   1:  PR[91,3] = PR[90,3] + 64.079;
   1:L PR[91] R[100]mm/sec CNT100;
   1:  PR[91,1] = PR[90,1] + 22.475;
   1:  PR[91,2] = PR[90,2] + -8.785;
   1:  PR[91,3] = PR[90,3] + 64.084;
   1:L PR[91] R[100]mm/sec CNT100;
   1:  PR[91,1] = PR[90,1] + 22.742;
   1:  PR[91,2] = PR[90,2] + -8.099;
   1:  PR[91,3] = PR[90,3] + 64.091;
   1:L PR[91] R[100]mm/sec CNT100;
   1:  PR[91,1] = PR[90,1] + 23.009;
   1:  PR[91,2] = PR[90,2] + -7.343;
   1:  PR[91,3] = PR[90,3] + 64.097;
   1:L PR[91] R[100]mm/sec CNT100;
   1:  PR[91,1] = PR[90,1] + 23.209;
   1:  PR[91,2] = PR[90,2] + -6.725;
   1:  PR[91,3] = PR[90,3] + 64.104;
   1:L PR[91] R[100]mm/sec CNT100;
   1:  PR[91,1] = PR[90,1] + 23.430;
   1:  PR[91,2] = PR[90,2] + -5.954;
   1:  PR[91,3] = PR[90,3] + 64.110;
   1:L PR[91] R[100]mm/sec CNT100;
   1:  PR[91,1] = PR[90,1] + 23.593;
   1:  PR[91,2] = PR[90,2] + -5.325;
   1:  PR[91,3] = PR[90,3] + 64.117;
   1:L PR[91] R[100]mm/sec CNT100;
   1:  PR[91,1] = PR[90,1] + 23.768;
   1:  PR[91,2] = PR[90,2] + -4.543;
   1:  PR[91,3] = PR[90,3] + 64.122;
   1:L PR[91] R[100]mm/sec CNT100;
   1:  PR[91,1] = PR[90,1] + 23.893;
   1:  PR[91,2] = PR[90,2] + -3.905;
   1:  PR[91,3] = PR[90,3] + 64.129;
   1:L PR[91] R[100]mm/sec CNT100;
   1:  PR[91,1] = PR[90,1] + 24.021;
   1:  PR[91,2] = PR[90,2] + -3.118;
   1:  PR[91,3] = PR[90,3] + 64.135;
   1:L PR[91] R[100]mm/sec CNT100;
   1:  PR[91,1] = PR[90,1] + 24.176;
   1:  PR[91,2] = PR[90,2] + -1.818;
   1:  PR[91,3] = PR[90,3] + 64.142;
   1:L PR[91] R[100]mm/sec CNT100;
   1:  PR[91,1] = PR[90,1] + 24.237;
   1:  PR[91,2] = PR[90,2] + -1.027;
   1:  PR[91,3] = PR[90,3] + 64.153;
   1:L PR[91] R[100]mm/sec CNT100;
   1:  PR[91,1] = PR[90,1] + 24.280;
   1:  PR[91,2] = PR[90,2] + 0.428;
   1:  PR[91,3] = PR[90,3] + 64.160;
   1:L PR[91] R[100]mm/sec CNT100;
   1:  PR[91,1] = PR[90,1] + 24.237;
   1:  PR[91,2] = PR[90,2] + 1.883;
   1:  PR[91,3] = PR[90,3] + 64.173;
   1:L PR[91] R[100]mm/sec CNT100;
   1:  PR[91,1] = PR[90,1] + 24.189;
   1:  PR[91,2] = PR[90,2] + 2.528;
   1:  PR[91,3] = PR[90,3] + 64.185;
   1:L PR[91] R[100]mm/sec CNT100;
   1:  PR[91,1] = PR[90,1] + 24.108;
   1:  PR[91,2] = PR[90,2] + 3.325;
   1:  PR[91,3] = PR[90,3] + 64.191;
   1:L PR[91] R[100]mm/sec CNT100;
   1:  PR[91,1] = PR[90,1] + 24.021;
   1:  PR[91,2] = PR[90,2] + 3.969;
   1:  PR[91,3] = PR[90,3] + 64.198;
   1:L PR[91] R[100]mm/sec CNT100;
   1:  PR[91,1] = PR[90,1] + 23.893;
   1:  PR[91,2] = PR[90,2] + 4.760;
   1:  PR[91,3] = PR[90,3] + 64.203;
   1:L PR[91] R[100]mm/sec CNT100;
   1:  PR[91,1] = PR[90,1] + 23.768;
   1:  PR[91,2] = PR[90,2] + 5.398;
   1:  PR[91,3] = PR[90,3] + 64.210;
   1:L PR[91] R[100]mm/sec CNT100;
   1:  PR[91,1] = PR[90,1] + 23.593;
   1:  PR[91,2] = PR[90,2] + 6.180;
   1:  PR[91,3] = PR[90,3] + 64.216;
   1:L PR[91] R[100]mm/sec CNT100;
   1:  PR[91,1] = PR[90,1] + 23.430;
   1:  PR[91,2] = PR[90,2] + 6.809;
   1:  PR[91,3] = PR[90,3] + 64.223;
   1:L PR[91] R[100]mm/sec CNT100;
   1:  PR[91,1] = PR[90,1] + 23.209;
   1:  PR[91,2] = PR[90,2] + 7.580;
   1:  PR[91,3] = PR[90,3] + 64.229;
   1:L PR[91] R[100]mm/sec CNT100;
   1:  PR[91,1] = PR[90,1] + 23.009;
   1:  PR[91,2] = PR[90,2] + 8.198;
   1:  PR[91,3] = PR[90,3] + 64.236;
   1:L PR[91] R[100]mm/sec CNT100;
   1:  PR[91,1] = PR[90,1] + 22.742;
   1:  PR[91,2] = PR[90,2] + 8.954;
   1:  PR[91,3] = PR[90,3] + 64.241;
   1:L PR[91] R[100]mm/sec CNT100;
   1:  PR[91,1] = PR[90,1] + 22.475;
   1:  PR[91,2] = PR[90,2] + 9.640;
   1:  PR[91,3] = PR[90,3] + 64.248;
   1:L PR[91] R[100]mm/sec CNT100;
   1:  PR[91,1] = PR[90,1] + 22.195;
   1:  PR[91,2] = PR[90,2] + 10.298;
   1:  PR[91,3] = PR[90,3] + 64.255;
   1:L PR[91] R[100]mm/sec CNT100;
   1:  PR[91,1] = PR[90,1] + 21.924;
   1:  PR[91,2] = PR[90,2] + 10.889;
   1:  PR[91,3] = PR[90,3] + 64.261;
   1:L PR[91] R[100]mm/sec CNT100;
   1:  PR[91,1] = PR[90,1] + 21.569;
   1:  PR[91,2] = PR[90,2] + 11.608;
   1:  PR[91,3] = PR[90,3] + 64.266;
   1:L PR[91] R[100]mm/sec CNT100;
   1:  PR[91,1] = PR[90,1] + 21.263;
   1:  PR[91,2] = PR[90,2] + 12.181;
   1:  PR[91,3] = PR[90,3] + 64.273;
   1:L PR[91] R[100]mm/sec CNT100;
   1:  PR[91,1] = PR[90,1] + 20.865;
   1:  PR[91,2] = PR[90,2] + 12.877;
   1:  PR[91,3] = PR[90,3] + 64.279;
   1:L PR[91] R[100]mm/sec CNT100;
   1:  PR[91,1] = PR[90,1] + 20.526;
   1:  PR[91,2] = PR[90,2] + 13.431;
   1:  PR[91,3] = PR[90,3] + 64.286;
   1:L PR[91] R[100]mm/sec CNT100;
   1:  PR[91,1] = PR[90,1] + 20.088;
   1:  PR[91,2] = PR[90,2] + 14.103;
   1:  PR[91,3] = PR[90,3] + 64.292;
   1:L PR[91] R[100]mm/sec CNT100;
   1:  PR[91,1] = PR[90,1] + 19.667;
   1:  PR[91,2] = PR[90,2] + 14.705;
   1:  PR[91,3] = PR[90,3] + 64.298;
   1:L PR[91] R[100]mm/sec CNT100;
   1:  PR[91,1] = PR[90,1] + 18.834;
   1:  PR[91,2] = PR[90,2] + 15.793;
   1:  PR[91,3] = PR[90,3] + 64.305;
   1:L PR[91] R[100]mm/sec CNT100;
   1:  PR[91,1] = PR[90,1] + 18.322;
   1:  PR[91,2] = PR[90,2] + 16.405;
   1:  PR[91,3] = PR[90,3] + 64.317;
   1:L PR[91] R[100]mm/sec CNT100;
   1:  PR[91,1] = PR[90,1] + 17.890;
   1:  PR[91,2] = PR[90,2] + 16.890;
   1:  PR[91,3] = PR[90,3] + 64.324;
   1:L PR[91] R[100]mm/sec CNT100;
   1:  PR[91,1] = PR[90,1] + 17.342;
   1:  PR[91,2] = PR[90,2] + 17.470;
   1:  PR[91,3] = PR[90,3] + 64.329;
   1:L PR[91] R[100]mm/sec CNT100;
   1:  PR[91,1] = PR[90,1] + 16.339;
   1:  PR[91,2] = PR[90,2] + 18.441;
   1:  PR[91,3] = PR[90,3] + 64.336;
   1:L PR[91] R[100]mm/sec CNT100;
   1:  PR[91,1] = PR[90,1] + 15.830;
   1:  PR[91,2] = PR[90,2] + 18.893;
   1:  PR[91,3] = PR[90,3] + 64.348;
   1:L PR[91] R[100]mm/sec CNT100;
   1:  PR[91,1] = PR[90,1] + 15.235;
   1:  PR[91,2] = PR[90,2] + 19.390;
   1:  PR[91,3] = PR[90,3] + 64.354;
   1:L PR[91] R[100]mm/sec CNT100;
   1:  PR[91,1] = PR[90,1] + 14.747;
   1:  PR[91,2] = PR[90,2] + 19.775;
   1:  PR[91,3] = PR[90,3] + 64.361;
   1:L PR[91] R[100]mm/sec CNT100;
   1:  PR[91,1] = PR[90,1] + 14.129;
   1:  PR[91,2] = PR[90,2] + 20.234;
   1:  PR[91,3] = PR[90,3] + 64.366;
   1:L PR[91] R[100]mm/sec CNT100;
   1:  PR[91,1] = PR[90,1] + 13.076;
   1:  PR[91,2] = PR[90,2] + 20.951;
   1:  PR[91,3] = PR[90,3] + 64.373;
   1:L PR[91] R[100]mm/sec CNT100;
   1:  PR[91,1] = PR[90,1] + 12.442;
   1:  PR[91,2] = PR[90,2] + 21.345;
   1:  PR[91,3] = PR[90,3] + 64.384;
   1:L PR[91] R[100]mm/sec CNT100;
   1:  PR[91,1] = PR[90,1] + 11.218;
   1:  PR[91,2] = PR[90,2] + 22.033;
   1:  PR[91,3] = PR[90,3] + 64.391;
   1:L PR[91] R[100]mm/sec CNT100;
   1:  PR[91,1] = PR[90,1] + 10.609;
   1:  PR[91,2] = PR[90,2] + 22.342;
   1:  PR[91,3] = PR[90,3] + 64.403;
   1:L PR[91] R[100]mm/sec CNT100;
   1:  PR[91,1] = PR[90,1] + 9.972;
   1:  PR[91,2] = PR[90,2] + 22.643;
   1:  PR[91,3] = PR[90,3] + 64.409;
   1:L PR[91] R[100]mm/sec CNT100;
   1:  PR[91,1] = PR[90,1] + 8.677;
   1:  PR[91,2] = PR[90,2] + 23.187;
   1:  PR[91,3] = PR[90,3] + 64.415;
   1:L PR[91] R[100]mm/sec CNT100;
   1:  PR[91,1] = PR[90,1] + 8.017;
   1:  PR[91,2] = PR[90,2] + 23.431;
   1:  PR[91,3] = PR[90,3] + 64.427;
   1:L PR[91] R[100]mm/sec CNT100;
   1:  PR[91,1] = PR[90,1] + 6.765;
   1:  PR[91,2] = PR[90,2] + 23.836;
   1:  PR[91,3] = PR[90,3] + 64.433;
   1:L PR[91] R[100]mm/sec CNT100;
   1:  PR[91,1] = PR[90,1] + 6.027;
   1:  PR[91,2] = PR[90,2] + 24.040;
   1:  PR[91,3] = PR[90,3] + 64.445;
   1:L PR[91] R[100]mm/sec CNT100;
   1:  PR[91,1] = PR[90,1] + 4.710;
   1:  PR[91,2] = PR[90,2] + 24.345;
   1:  PR[91,3] = PR[90,3] + 64.451;
   1:L PR[91] R[100]mm/sec CNT100;
   1:  PR[91,1] = PR[90,1] + 4.050;
   1:  PR[91,2] = PR[90,2] + 24.468;
   1:  PR[91,3] = PR[90,3] + 64.463;
   1:L PR[91] R[100]mm/sec CNT100;
   1:  PR[91,1] = PR[90,1] + 3.290;
   1:  PR[91,2] = PR[90,2] + 24.588;
   1:  PR[91,3] = PR[90,3] + 64.469;
   1:L PR[91] R[100]mm/sec CNT100;
   1:  PR[91,1] = PR[90,1] + 1.949;
   1:  PR[91,2] = PR[90,2] + 24.739;
   1:  PR[91,3] = PR[90,3] + 64.475;
   1:L PR[91] R[100]mm/sec CNT100;
   1:  PR[91,1] = PR[90,1] + 0.649;
   1:  PR[91,2] = PR[90,2] + 24.814;
   1:  PR[91,3] = PR[90,3] + 64.487;
   1:L PR[91] R[100]mm/sec CNT100;
   1:  PR[91,1] = PR[90,1] + -0.121;
   1:  PR[91,2] = PR[90,2] + 24.827;
   1:  PR[91,3] = PR[90,3] + 64.498;
   1:L PR[91] R[100]mm/sec CNT100;
   1:  PR[91,1] = PR[90,1] + -0.841;
   1:  PR[91,2] = PR[90,2] + 24.817;
   1:  PR[91,3] = PR[90,3] + 64.505;
   1:L PR[91] R[100]mm/sec CNT100;
   1:  PR[91,1] = PR[90,1] + -1.512;
   1:  PR[91,2] = PR[90,2] + 24.788;
   1:  PR[91,3] = PR[90,3] + 64.511;
   1:L PR[91] R[100]mm/sec CNT100;
   1:  PR[91,1] = PR[90,1] + -2.912;
   1:  PR[91,2] = PR[90,2] + 24.667;
   1:  PR[91,3] = PR[90,3] + 64.517;
   1:L PR[91] R[100]mm/sec CNT100;
   1:  PR[91,1] = PR[90,1] + -3.618;
   1:  PR[91,2] = PR[90,2] + 24.575;
   1:  PR[91,3] = PR[90,3] + 64.529;
   1:L PR[91] R[100]mm/sec CNT100;
   1:  PR[91,1] = PR[90,1] + -4.905;
   1:  PR[91,2] = PR[90,2] + 24.353;
   1:  PR[91,3] = PR[90,3] + 64.536;
   1:L PR[91] R[100]mm/sec CNT100;
   1:  PR[91,1] = PR[90,1] + -5.654;
   1:  PR[91,2] = PR[90,2] + 24.191;
   1:  PR[91,3] = PR[90,3] + 64.547;
   1:L PR[91] R[100]mm/sec CNT100;
   1:  PR[91,1] = PR[90,1] + -6.967;
   1:  PR[91,2] = PR[90,2] + 23.847;
   1:  PR[91,3] = PR[90,3] + 64.553;
   1:L PR[91] R[100]mm/sec CNT100;
   1:  PR[91,1] = PR[90,1] + -7.599;
   1:  PR[91,2] = PR[90,2] + 23.653;
   1:  PR[91,3] = PR[90,3] + 64.565;
   1:L PR[91] R[100]mm/sec CNT100;
   1:  PR[91,1] = PR[90,1] + -8.919;
   1:  PR[91,2] = PR[90,2] + 23.185;
   1:  PR[91,3] = PR[90,3] + 64.571;
   1:L PR[91] R[100]mm/sec CNT100;
   1:  PR[91,1] = PR[90,1] + -10.180;
   1:  PR[91,2] = PR[90,2] + 22.656;
   1:  PR[91,3] = PR[90,3] + 64.583;
   1:L PR[91] R[100]mm/sec CNT100;
   1:  PR[91,1] = PR[90,1] + -11.461;
   1:  PR[91,2] = PR[90,2] + 22.031;
   1:  PR[91,3] = PR[90,3] + 64.595;
   1:L PR[91] R[100]mm/sec CNT100;
   1:  PR[91,1] = PR[90,1] + -12.678;
   1:  PR[91,2] = PR[90,2] + 21.347;
   1:  PR[91,3] = PR[90,3] + 64.607;
   1:L PR[91] R[100]mm/sec CNT100;
   1:  PR[91,1] = PR[90,1] + -13.854;
   1:  PR[91,2] = PR[90,2] + 20.594;
   1:  PR[91,3] = PR[90,3] + 64.619;
   1:L PR[91] R[100]mm/sec CNT100;
   1:  PR[91,1] = PR[90,1] + -14.988;
   1:  PR[91,2] = PR[90,2] + 19.774;
   1:  PR[91,3] = PR[90,3] + 64.632;
   1:L PR[91] R[100]mm/sec CNT100;
   1:  PR[91,1] = PR[90,1] + -15.529;
   1:  PR[91,2] = PR[90,2] + 19.346;
   1:  PR[91,3] = PR[90,3] + 64.644;
   1:L PR[91] R[100]mm/sec CNT100;
   1:  PR[91,1] = PR[90,1] + -16.536;
   1:  PR[91,2] = PR[90,2] + 18.478;
   1:  PR[91,3] = PR[90,3] + 64.650;
   1:L PR[91] R[100]mm/sec CNT100;
   1:  PR[91,1] = PR[90,1] + -17.118;
   1:  PR[91,2] = PR[90,2] + 17.932;
   1:  PR[91,3] = PR[90,3] + 64.661;
   1:L PR[91] R[100]mm/sec CNT100;
   1:  PR[91,1] = PR[90,1] + -17.577;
   1:  PR[91,2] = PR[90,2] + 17.473;
   1:  PR[91,3] = PR[90,3] + 64.668;
   1:L PR[91] R[100]mm/sec CNT100;
   1:  PR[91,1] = PR[90,1] + -18.125;
   1:  PR[91,2] = PR[90,2] + 16.894;
   1:  PR[91,3] = PR[90,3] + 64.674;
   1:L PR[91] R[100]mm/sec CNT100;
   1:  PR[91,1] = PR[90,1] + -19.010;
   1:  PR[91,2] = PR[90,2] + 15.869;
   1:  PR[91,3] = PR[90,3] + 64.681;
   1:L PR[91] R[100]mm/sec CNT100;
   1:  PR[91,1] = PR[90,1] + -19.478;
   1:  PR[91,2] = PR[90,2] + 15.280;
   1:  PR[91,3] = PR[90,3] + 64.692;
   1:L PR[91] R[100]mm/sec CNT100;
   1:  PR[91,1] = PR[90,1] + -19.955;
   1:  PR[91,2] = PR[90,2] + 14.636;
   1:  PR[91,3] = PR[90,3] + 64.699;
   1:L PR[91] R[100]mm/sec CNT100;
   1:  PR[91,1] = PR[90,1] + -20.326;
   1:  PR[91,2] = PR[90,2] + 14.103;
   1:  PR[91,3] = PR[90,3] + 64.706;
   1:L PR[91] R[100]mm/sec CNT100;
   1:  PR[91,1] = PR[90,1] + -20.764;
   1:  PR[91,2] = PR[90,2] + 13.432;
   1:  PR[91,3] = PR[90,3] + 64.712;
   1:L PR[91] R[100]mm/sec CNT100;
   1:  PR[91,1] = PR[90,1] + -21.104;
   1:  PR[91,2] = PR[90,2] + 12.878;
   1:  PR[91,3] = PR[90,3] + 64.719;
   1:L PR[91] R[100]mm/sec CNT100;
   1:  PR[91,1] = PR[90,1] + -21.488;
   1:  PR[91,2] = PR[90,2] + 12.206;
   1:  PR[91,3] = PR[90,3] + 64.724;
   1:L PR[91] R[100]mm/sec CNT100;
   1:  PR[91,1] = PR[90,1] + -21.794;
   1:  PR[91,2] = PR[90,2] + 11.632;
   1:  PR[91,3] = PR[90,3] + 64.731;
   1:L PR[91] R[100]mm/sec CNT100;
   1:  PR[91,1] = PR[90,1] + -22.160;
   1:  PR[91,2] = PR[90,2] + 10.893;
   1:  PR[91,3] = PR[90,3] + 64.737;
   1:L PR[91] R[100]mm/sec CNT100;
   1:  PR[91,1] = PR[90,1] + -22.689;
   1:  PR[91,2] = PR[90,2] + 9.695;
   1:  PR[91,3] = PR[90,3] + 64.744;
   1:L PR[91] R[100]mm/sec CNT100;
   1:  PR[91,1] = PR[90,1] + -22.981;
   1:  PR[91,2] = PR[90,2] + 8.953;
   1:  PR[91,3] = PR[90,3] + 64.755;
   1:L PR[91] R[100]mm/sec CNT100;
   1:  PR[91,1] = PR[90,1] + -23.248;
   1:  PR[91,2] = PR[90,2] + 8.199;
   1:  PR[91,3] = PR[90,3] + 64.762;
   1:L PR[91] R[100]mm/sec CNT100;
   1:  PR[91,1] = PR[90,1] + -23.447;
   1:  PR[91,2] = PR[90,2] + 7.580;
   1:  PR[91,3] = PR[90,3] + 64.769;
   1:L PR[91] R[100]mm/sec CNT100;
   1:  PR[91,1] = PR[90,1] + -23.669;
   1:  PR[91,2] = PR[90,2] + 6.810;
   1:  PR[91,3] = PR[90,3] + 64.775;
   1:L PR[91] R[100]mm/sec CNT100;
   1:  PR[91,1] = PR[90,1] + -23.831;
   1:  PR[91,2] = PR[90,2] + 6.181;
   1:  PR[91,3] = PR[90,3] + 64.782;
   1:L PR[91] R[100]mm/sec CNT100;
   1:  PR[91,1] = PR[90,1] + -24.006;
   1:  PR[91,2] = PR[90,2] + 5.402;
   1:  PR[91,3] = PR[90,3] + 64.787;
   1:L PR[91] R[100]mm/sec CNT100;
   1:  PR[91,1] = PR[90,1] + -24.238;
   1:  PR[91,2] = PR[90,2] + 4.113;
   1:  PR[91,3] = PR[90,3] + 64.794;
   1:L PR[91] R[100]mm/sec CNT100;
   1:  PR[91,1] = PR[90,1] + -24.347;
   1:  PR[91,2] = PR[90,2] + 3.324;
   1:  PR[91,3] = PR[90,3] + 64.805;
   1:L PR[91] R[100]mm/sec CNT100;
   1:  PR[91,1] = PR[90,1] + -24.428;
   1:  PR[91,2] = PR[90,2] + 2.528;
   1:  PR[91,3] = PR[90,3] + 64.812;
   1:L PR[91] R[100]mm/sec CNT100;
   1:  PR[91,1] = PR[90,1] + -24.476;
   1:  PR[91,2] = PR[90,2] + 1.883;
   1:  PR[91,3] = PR[90,3] + 64.819;
   1:L PR[91] R[100]mm/sec CNT100;
   1:  PR[91,1] = PR[90,1] + -24.519;
   1:  PR[91,2] = PR[90,2] + 0.428;
   1:  PR[91,3] = PR[90,3] + 64.825;
   1:L PR[91] R[100]mm/sec CNT100;
   1:  PR[91,1] = PR[90,1] + -24.476;
   1:  PR[91,2] = PR[90,2] + -1.028;
   1:  PR[91,3] = PR[90,3] + 64.838;
   1:L PR[91] R[100]mm/sec CNT100;
   1:  PR[91,1] = PR[90,1] + -24.428;
   1:  PR[91,2] = PR[90,2] + -1.673;
   1:  PR[91,3] = PR[90,3] + 64.850;
   1:L PR[91] R[100]mm/sec CNT100;
   1:  PR[91,1] = PR[90,1] + -24.346;
   1:  PR[91,2] = PR[90,2] + -2.470;
   1:  PR[91,3] = PR[90,3] + 64.856;
   1:L PR[91] R[100]mm/sec CNT100;
   1:  PR[91,1] = PR[90,1] + -24.260;
   1:  PR[91,2] = PR[90,2] + -3.114;
   1:  PR[91,3] = PR[90,3] + 64.863;
   1:L PR[91] R[100]mm/sec CNT100;
   1:  PR[91,1] = PR[90,1] + -24.131;
   1:  PR[91,2] = PR[90,2] + -3.905;
   1:  PR[91,3] = PR[90,3] + 64.868;
   1:L PR[91] R[100]mm/sec CNT100;
   1:  PR[91,1] = PR[90,1] + -24.007;
   1:  PR[91,2] = PR[90,2] + -4.543;
   1:  PR[91,3] = PR[90,3] + 64.875;
   1:L PR[91] R[100]mm/sec CNT100;
   1:  PR[91,1] = PR[90,1] + -23.832;
   1:  PR[91,2] = PR[90,2] + -5.321;
   1:  PR[91,3] = PR[90,3] + 64.881;
   1:L PR[91] R[100]mm/sec CNT100;
   1:  PR[91,1] = PR[90,1] + -23.484;
   1:  PR[91,2] = PR[90,2] + -6.594;
   1:  PR[91,3] = PR[90,3] + 64.888;
   1:L PR[91] R[100]mm/sec CNT100;
   1:  PR[91,1] = PR[90,1] + -23.446;
   1:  PR[91,2] = PR[90,2] + -6.728;
   1:  PR[91,3] = PR[90,3] + 64.899;
   1:L PR[91] R[100]mm/sec CNT100;
   1:  PR[91,1] = PR[90,1] + -23.248;
   1:  PR[91,2] = PR[90,2] + -7.344;
   1:  PR[91,3] = PR[90,3] + 64.901;
   1:L PR[91] R[100]mm/sec CNT100;
   1:  PR[91,1] = PR[90,1] + -22.981;
   1:  PR[91,2] = PR[90,2] + -8.100;
   1:  PR[91,3] = PR[90,3] + 64.906;
   1:L PR[91] R[100]mm/sec CNT100;
   1:  PR[91,1] = PR[90,1] + -22.745;
   1:  PR[91,2] = PR[90,2] + -8.705;
   1:  PR[91,3] = PR[90,3] + 64.913;
   1:L PR[91] R[100]mm/sec CNT100;
   1:  PR[91,1] = PR[90,1] + -22.433;
   1:  PR[91,2] = PR[90,2] + -9.444;
   1:  PR[91,3] = PR[90,3] + 64.919;
   1:L PR[91] R[100]mm/sec CNT100;
   1:  PR[91,1] = PR[90,1] + -22.162;
   1:  PR[91,2] = PR[90,2] + -10.034;
   1:  PR[91,3] = PR[90,3] + 64.926;
   1:L PR[91] R[100]mm/sec CNT100;
   1:  PR[91,1] = PR[90,1] + -21.807;
   1:  PR[91,2] = PR[90,2] + -10.753;
   1:  PR[91,3] = PR[90,3] + 64.931;
   1:L PR[91] R[100]mm/sec CNT100;
   1:  PR[91,1] = PR[90,1] + -21.501;
   1:  PR[91,2] = PR[90,2] + -11.326;
   1:  PR[91,3] = PR[90,3] + 64.938;
   1:L PR[91] R[100]mm/sec CNT100;
   1:  PR[91,1] = PR[90,1] + -21.104;
   1:  PR[91,2] = PR[90,2] + -12.023;
   1:  PR[91,3] = PR[90,3] + 64.944;
   1:L PR[91] R[100]mm/sec CNT100;
   1:  PR[91,1] = PR[90,1] + -20.764;
   1:  PR[91,2] = PR[90,2] + -12.576;
   1:  PR[91,3] = PR[90,3] + 64.951;
   1:L PR[91] R[100]mm/sec CNT100;
   1:  PR[91,1] = PR[90,1] + -20.326;
   1:  PR[91,2] = PR[90,2] + -13.248;
   1:  PR[91,3] = PR[90,3] + 64.957;
   1:L PR[91] R[100]mm/sec CNT100;
   1:  PR[91,1] = PR[90,1] + -19.955;
   1:  PR[91,2] = PR[90,2] + -13.781;
   1:  PR[91,3] = PR[90,3] + 64.963;
   1:L PR[91] R[100]mm/sec CNT100;
   1:  PR[91,1] = PR[90,1] + -19.478;
   1:  PR[91,2] = PR[90,2] + -14.425;
   1:  PR[91,3] = PR[90,3] + 64.969;
   1:L PR[91] R[100]mm/sec CNT100;
   1:  PR[91,1] = PR[90,1] + -19.010;
   1:  PR[91,2] = PR[90,2] + -15.014;
   1:  PR[91,3] = PR[90,3] + 64.976;
   1:L PR[91] R[100]mm/sec CNT100;
   1:  PR[91,1] = PR[90,1] + -18.125;
   1:  PR[91,2] = PR[90,2] + -16.038;
   1:  PR[91,3] = PR[90,3] + 64.983;
   1:L PR[91] R[100]mm/sec CNT100;
   1:  PR[91,1] = PR[90,1] + -17.577;
   1:  PR[91,2] = PR[90,2] + -16.618;
   1:  PR[91,3] = PR[90,3] + 64.994;
   1:L PR[91] R[100]mm/sec CNT100;
   1:  PR[91,1] = PR[90,1] + -17.118;
   1:  PR[91,2] = PR[90,2] + -17.077;
   1:  PR[91,3] = PR[90,3] + 65.001;
   1:L PR[91] R[100]mm/sec CNT100;
   1:  PR[91,1] = PR[90,1] + -16.536;
   1:  PR[91,2] = PR[90,2] + -17.623;
   1:  PR[91,3] = PR[90,3] + 65.007;
   1:L PR[91] R[100]mm/sec CNT100;
   1:  PR[91,1] = PR[90,1] + -15.529;
   1:  PR[91,2] = PR[90,2] + -18.490;
   1:  PR[91,3] = PR[90,3] + 65.014;
   1:L PR[91] R[100]mm/sec CNT100;
   1:  PR[91,1] = PR[90,1] + -14.988;
   1:  PR[91,2] = PR[90,2] + -18.918;
   1:  PR[91,3] = PR[90,3] + 65.025;
   1:L PR[91] R[100]mm/sec CNT100;
   1:  PR[91,1] = PR[90,1] + -13.854;
   1:  PR[91,2] = PR[90,2] + -19.739;
   1:  PR[91,3] = PR[90,3] + 65.031;
   1:L PR[91] R[100]mm/sec CNT100;
   1:  PR[91,1] = PR[90,1] + -12.684;
   1:  PR[91,2] = PR[90,2] + -20.488;
   1:  PR[91,3] = PR[90,3] + 65.043;
   1:L PR[91] R[100]mm/sec CNT100;
   1:  PR[91,1] = PR[90,1] + -11.461;
   1:  PR[91,2] = PR[90,2] + -21.176;
   1:  PR[91,3] = PR[90,3] + 65.056;
   1:L PR[91] R[100]mm/sec CNT100;
   1:  PR[91,1] = PR[90,1] + -10.207;
   1:  PR[91,2] = PR[90,2] + -21.789;
   1:  PR[91,3] = PR[90,3] + 65.068;
   1:L PR[91] R[100]mm/sec CNT100;
   1:  PR[91,1] = PR[90,1] + -8.919;
   1:  PR[91,2] = PR[90,2] + -22.330;
   1:  PR[91,3] = PR[90,3] + 65.080;
   1:L PR[91] R[100]mm/sec CNT100;
   1:  PR[91,1] = PR[90,1] + -7.599;
   1:  PR[91,2] = PR[90,2] + -22.797;
   1:  PR[91,3] = PR[90,3] + 65.092;
   1:L PR[91] R[100]mm/sec CNT100;
   1:  PR[91,1] = PR[90,1] + -6.967;
   1:  PR[91,2] = PR[90,2] + -22.992;
   1:  PR[91,3] = PR[90,3] + 65.104;
   1:L PR[91] R[100]mm/sec CNT100;
   1:  PR[91,1] = PR[90,1] + -5.654;
   1:  PR[91,2] = PR[90,2] + -23.336;
   1:  PR[91,3] = PR[90,3] + 65.110;
   1:L PR[91] R[100]mm/sec CNT100;
   1:  PR[91,1] = PR[90,1] + -4.905;
   1:  PR[91,2] = PR[90,2] + -23.498;
   1:  PR[91,3] = PR[90,3] + 65.122;
   1:L PR[91] R[100]mm/sec CNT100;
   1:  PR[91,1] = PR[90,1] + -3.618;
   1:  PR[91,2] = PR[90,2] + -23.720;
   1:  PR[91,3] = PR[90,3] + 65.128;
   1:L PR[91] R[100]mm/sec CNT100;
   1:  PR[91,1] = PR[90,1] + -2.908;
   1:  PR[91,2] = PR[90,2] + -23.812;
   1:  PR[91,3] = PR[90,3] + 65.140;
   1:L PR[91] R[100]mm/sec CNT100;
   1:  PR[91,1] = PR[90,1] + -2.288;
   1:  PR[91,2] = PR[90,2] + -23.874;
   1:  PR[91,3] = PR[90,3] + 65.146;
   1:L PR[91] R[100]mm/sec CNT100;
   1:  PR[91,1] = PR[90,1] + -1.515;
   1:  PR[91,2] = PR[90,2] + -23.932;
   1:  PR[91,3] = PR[90,3] + 65.151;
   1:L PR[91] R[100]mm/sec CNT100;
   1:  PR[91,1] = PR[90,1] + -0.841;
   1:  PR[91,2] = PR[90,2] + -23.962;
   1:  PR[91,3] = PR[90,3] + 65.158;
   1:L PR[91] R[100]mm/sec CNT100;
   1:  PR[91,1] = PR[90,1] + -0.124;
   1:  PR[91,2] = PR[90,2] + -23.972;
   1:  PR[91,3] = PR[90,3] + 65.164;
   1:L PR[91] R[100]mm/sec CNT100;
   1:  PR[91] = PR[90];
   1:  PR[91,1] = PR[90,1] + 1.301;
   1:  PR[91,2] = PR[90,2] + -23.931;
   1:  PR[91,3] = PR[90,3] + 66.500;
   1:L PR[91] R[100]mm/sec CNT100;
   1:  PR[91,1] = PR[90,1] + 1.921;
   1:  PR[91,2] = PR[90,2] + -23.887;
   1:  PR[91,3] = PR[90,3] + 65.179;
   1:L PR[91] R[100]mm/sec CNT100;
   1:  PR[91,1] = PR[90,1] + 2.710;
   1:  PR[91,2] = PR[90,2] + -23.807;
   1:  PR[91,3] = PR[90,3] + 65.184;
   1:L PR[91] R[100]mm/sec CNT100;
   1:  PR[91,1] = PR[90,1] + 4.122;
   1:  PR[91,2] = PR[90,2] + -23.601;
   1:  PR[91,3] = PR[90,3] + 65.191;
   1:L PR[91] R[100]mm/sec CNT100;
   1:  PR[91,1] = PR[90,1] + 4.733;
   1:  PR[91,2] = PR[90,2] + -23.485;
   1:  PR[91,3] = PR[90,3] + 65.203;
   1:L PR[91] R[100]mm/sec CNT100;
   1:  PR[91,1] = PR[90,1] + 5.932;
   1:  PR[91,2] = PR[90,2] + -23.209;
   1:  PR[91,3] = PR[90,3] + 65.209;
   1:L PR[91] R[100]mm/sec CNT100;
   1:  PR[91,1] = PR[90,1] + 7.303;
   1:  PR[91,2] = PR[90,2] + -22.816;
   1:  PR[91,3] = PR[90,3] + 65.219;
   1:L PR[91] R[100]mm/sec CNT100;
   1:  PR[91,1] = PR[90,1] + 7.926;
   1:  PR[91,2] = PR[90,2] + -22.607;
   1:  PR[91,3] = PR[90,3] + 65.232;
   1:L PR[91] R[100]mm/sec CNT100;
   1:  PR[91,1] = PR[90,1] + 8.635;
   1:  PR[91,2] = PR[90,2] + -22.348;
   1:  PR[91,3] = PR[90,3] + 65.237;
   1:L PR[91] R[100]mm/sec CNT100;
   1:  PR[91,1] = PR[90,1] + 9.543;
   1:  PR[91,2] = PR[90,2] + -21.976;
   1:  PR[91,3] = PR[90,3] + 65.244;
   1:L PR[91] R[100]mm/sec CNT100;
   1:  PR[91,1] = PR[90,1] + 10.623;
   1:  PR[91,2] = PR[90,2] + -21.480;
   1:  PR[91,3] = PR[90,3] + 65.252;
   1:L PR[91] R[100]mm/sec CNT100;
   1:  PR[91,1] = PR[90,1] + 11.608;
   1:  PR[91,2] = PR[90,2] + -20.967;
   1:  PR[91,3] = PR[90,3] + 65.263;
   1:L PR[91] R[100]mm/sec CNT100;
   1:  PR[91,1] = PR[90,1] + 12.457;
   1:  PR[91,2] = PR[90,2] + -20.481;
   1:  PR[91,3] = PR[90,3] + 65.272;
   1:L PR[91] R[100]mm/sec CNT100;
   1:  PR[91,1] = PR[90,1] + 13.594;
   1:  PR[91,2] = PR[90,2] + -19.754;
   1:  PR[91,3] = PR[90,3] + 65.281;
   1:L PR[91] R[100]mm/sec CNT100;
   1:  PR[91,1] = PR[90,1] + 14.800;
   1:  PR[91,2] = PR[90,2] + -18.879;
   1:  PR[91,3] = PR[90,3] + 65.293;
   1:L PR[91] R[100]mm/sec CNT100;
   1:  PR[91,1] = PR[90,1] + 15.899;
   1:  PR[91,2] = PR[90,2] + -17.977;
   1:  PR[91,3] = PR[90,3] + 65.305;
   1:L PR[91] R[100]mm/sec CNT100;
   1:  PR[91,1] = PR[90,1] + 16.730;
   1:  PR[91,2] = PR[90,2] + -17.219;
   1:  PR[91,3] = PR[90,3] + 65.318;
   1:L PR[91] R[100]mm/sec CNT100;
   1:  PR[91,1] = PR[90,1] + 17.276;
   1:  PR[91,2] = PR[90,2] + -16.682;
   1:  PR[91,3] = PR[90,3] + 65.328;
   1:L PR[91] R[100]mm/sec CNT100;
   1:  PR[91,1] = PR[90,1] + 18.269;
   1:  PR[91,2] = PR[90,2] + -15.609;
   1:  PR[91,3] = PR[90,3] + 65.334;
   1:L PR[91] R[100]mm/sec CNT100;
   1:  PR[91,1] = PR[90,1] + 19.198;
   1:  PR[91,2] = PR[90,2] + -14.478;
   1:  PR[91,3] = PR[90,3] + 65.347;
   1:L PR[91] R[100]mm/sec CNT100;
   1:  PR[91,1] = PR[90,1] + 19.601;
   1:  PR[91,2] = PR[90,2] + -13.940;
   1:  PR[91,3] = PR[90,3] + 65.360;
   1:L PR[91] R[100]mm/sec CNT100;
   1:  PR[91,1] = PR[90,1] + 20.050;
   1:  PR[91,2] = PR[90,2] + -13.304;
   1:  PR[91,3] = PR[90,3] + 65.365;
   1:L PR[91] R[100]mm/sec CNT100;
   1:  PR[91,1] = PR[90,1] + 20.595;
   1:  PR[91,2] = PR[90,2] + -12.465;
   1:  PR[91,3] = PR[90,3] + 65.372;
   1:L PR[91] R[100]mm/sec CNT100;
   1:  PR[91,1] = PR[90,1] + 21.062;
   1:  PR[91,2] = PR[90,2] + -11.675;
   1:  PR[91,3] = PR[90,3] + 65.381;
   1:L PR[91] R[100]mm/sec CNT100;
   1:  PR[91,1] = PR[90,1] + 21.544;
   1:  PR[91,2] = PR[90,2] + -10.800;
   1:  PR[91,3] = PR[90,3] + 65.389;
   1:L PR[91] R[100]mm/sec CNT100;
   1:  PR[91,1] = PR[90,1] + 22.177;
   1:  PR[91,2] = PR[90,2] + -9.483;
   1:  PR[91,3] = PR[90,3] + 65.397;
   1:L PR[91] R[100]mm/sec CNT100;
   1:  PR[91,1] = PR[90,1] + 22.564;
   1:  PR[91,2] = PR[90,2] + -8.559;
   1:  PR[91,3] = PR[90,3] + 65.410;
   1:L PR[91] R[100]mm/sec CNT100;
   1:  PR[91,1] = PR[90,1] + 22.728;
   1:  PR[91,2] = PR[90,2] + -8.138;
   1:  PR[91,3] = PR[90,3] + 65.419;
   1:L PR[91] R[100]mm/sec CNT100;
   1:  PR[91,1] = PR[90,1] + 23.058;
   1:  PR[91,2] = PR[90,2] + -7.193;
   1:  PR[91,3] = PR[90,3] + 65.423;
   1:L PR[91] R[100]mm/sec CNT100;
   1:  PR[91,1] = PR[90,1] + 23.327;
   1:  PR[91,2] = PR[90,2] + -6.316;
   1:  PR[91,3] = PR[90,3] + 65.431;
   1:L PR[91] R[100]mm/sec CNT100;
   1:  PR[91,1] = PR[90,1] + 23.586;
   1:  PR[91,2] = PR[90,2] + -5.352;
   1:  PR[91,3] = PR[90,3] + 65.439;
   1:L PR[91] R[100]mm/sec CNT100;
   1:  PR[91,1] = PR[90,1] + 23.889;
   1:  PR[91,2] = PR[90,2] + -3.923;
   1:  PR[91,3] = PR[90,3] + 65.448;
   1:L PR[91] R[100]mm/sec CNT100;
   1:  PR[91,1] = PR[90,1] + 24.106;
   1:  PR[91,2] = PR[90,2] + -2.481;
   1:  PR[91,3] = PR[90,3] + 65.461;
   1:L PR[91] R[100]mm/sec CNT100;
   1:  PR[91,1] = PR[90,1] + 24.203;
   1:  PR[91,2] = PR[90,2] + -1.490;
   1:  PR[91,3] = PR[90,3] + 65.473;
   1:L PR[91] R[100]mm/sec CNT100;
   1:  PR[91,1] = PR[90,1] + 24.257;
   1:  PR[91,2] = PR[90,2] + -0.574;
   1:  PR[91,3] = PR[90,3] + 65.482;
   1:L PR[91] R[100]mm/sec CNT100;
   1:  PR[91,1] = PR[90,1] + 24.281;
   1:  PR[91,2] = PR[90,2] + 0.430;
   1:  PR[91,3] = PR[90,3] + 65.490;
   1:L PR[91] R[100]mm/sec CNT100;
   1:  PR[91,1] = PR[90,1] + 24.274;
   1:  PR[91,2] = PR[90,2] + 0.882;
   1:  PR[91,3] = PR[90,3] + 65.499;
   1:L PR[91] R[100]mm/sec CNT100;
   1:  PR[91,1] = PR[90,1] + 24.237;
   1:  PR[91,2] = PR[90,2] + 1.885;
   1:  PR[91,3] = PR[90,3] + 65.503;
   1:L PR[91] R[100]mm/sec CNT100;
   1:  PR[91,1] = PR[90,1] + 24.106;
   1:  PR[91,2] = PR[90,2] + 3.339;
   1:  PR[91,3] = PR[90,3] + 65.511;
   1:L PR[91] R[100]mm/sec CNT100;
   1:  PR[91,1] = PR[90,1] + 23.889;
   1:  PR[91,2] = PR[90,2] + 4.783;
   1:  PR[91,3] = PR[90,3] + 65.524;
   1:L PR[91] R[100]mm/sec CNT100;
   1:  PR[91,1] = PR[90,1] + 23.802;
   1:  PR[91,2] = PR[90,2] + 5.225;
   1:  PR[91,3] = PR[90,3] + 65.537;
   1:L PR[91] R[100]mm/sec CNT100;
   1:  PR[91,1] = PR[90,1] + 23.587;
   1:  PR[91,2] = PR[90,2] + 6.203;
   1:  PR[91,3] = PR[90,3] + 65.541;
   1:L PR[91] R[100]mm/sec CNT100;
   1:  PR[91,1] = PR[90,1] + 23.199;
   1:  PR[91,2] = PR[90,2] + 7.611;
   1:  PR[91,3] = PR[90,3] + 65.549;
   1:L PR[91] R[100]mm/sec CNT100;
   1:  PR[91,1] = PR[90,1] + 22.727;
   1:  PR[91,2] = PR[90,2] + 8.994;
   1:  PR[91,3] = PR[90,3] + 65.562;
   1:L PR[91] R[100]mm/sec CNT100;
   1:  PR[91,1] = PR[90,1] + 22.448;
   1:  PR[91,2] = PR[90,2] + 9.703;
   1:  PR[91,3] = PR[90,3] + 65.575;
   1:L PR[91] R[100]mm/sec CNT100;
   1:  PR[91,1] = PR[90,1] + 21.984;
   1:  PR[91,2] = PR[90,2] + 10.758;
   1:  PR[91,3] = PR[90,3] + 65.581;
   1:L PR[91] R[100]mm/sec CNT100;
   1:  PR[91,1] = PR[90,1] + 21.545;
   1:  PR[91,2] = PR[90,2] + 11.652;
   1:  PR[91,3] = PR[90,3] + 65.591;
   1:L PR[91] R[100]mm/sec CNT100;
   1:  PR[91,1] = PR[90,1] + 20.835;
   1:  PR[91,2] = PR[90,2] + 12.928;
   1:  PR[91,3] = PR[90,3] + 65.600;
   1:L PR[91] R[100]mm/sec CNT100;
   1:  PR[91,1] = PR[90,1] + 20.048;
   1:  PR[91,2] = PR[90,2] + 14.161;
   1:  PR[91,3] = PR[90,3] + 65.613;
   1:L PR[91] R[100]mm/sec CNT100;
   1:  PR[91,1] = PR[90,1] + 19.603;
   1:  PR[91,2] = PR[90,2] + 14.793;
   1:  PR[91,3] = PR[90,3] + 65.625;
   1:L PR[91] R[100]mm/sec CNT100;
   1:  PR[91,1] = PR[90,1] + 18.910;
   1:  PR[91,2] = PR[90,2] + 15.698;
   1:  PR[91,3] = PR[90,3] + 65.632;
   1:L PR[91] R[100]mm/sec CNT100;
   1:  PR[91,1] = PR[90,1] + 18.271;
   1:  PR[91,2] = PR[90,2] + 16.462;
   1:  PR[91,3] = PR[90,3] + 65.642;
   1:L PR[91] R[100]mm/sec CNT100;
   1:  PR[91,1] = PR[90,1] + 17.276;
   1:  PR[91,2] = PR[90,2] + 17.537;
   1:  PR[91,3] = PR[90,3] + 65.650;
   1:L PR[91] R[100]mm/sec CNT100;
   1:  PR[91,1] = PR[90,1] + 16.728;
   1:  PR[91,2] = PR[90,2] + 18.076;
   1:  PR[91,3] = PR[90,3] + 65.663;
   1:L PR[91] R[100]mm/sec CNT100;
   1:  PR[91,1] = PR[90,1] + 16.230;
   1:  PR[91,2] = PR[90,2] + 18.539;
   1:  PR[91,3] = PR[90,3] + 65.670;
   1:L PR[91] R[100]mm/sec CNT100;
   1:  PR[91,1] = PR[90,1] + 15.145;
   1:  PR[91,2] = PR[90,2] + 19.462;
   1:  PR[91,3] = PR[90,3] + 65.676;
   1:L PR[91] R[100]mm/sec CNT100;
   1:  PR[91,1] = PR[90,1] + 14.011;
   1:  PR[91,2] = PR[90,2] + 20.318;
   1:  PR[91,3] = PR[90,3] + 65.688;
   1:L PR[91] R[100]mm/sec CNT100;
   1:  PR[91,1] = PR[90,1] + 13.227;
   1:  PR[91,2] = PR[90,2] + 20.851;
   1:  PR[91,3] = PR[90,3] + 65.700;
   1:L PR[91] R[100]mm/sec CNT100;
   1:  PR[91,1] = PR[90,1] + 12.460;
   1:  PR[91,2] = PR[90,2] + 21.334;
   1:  PR[91,3] = PR[90,3] + 65.709;
   1:L PR[91] R[100]mm/sec CNT100;
   1:  PR[91,1] = PR[90,1] + 11.217;
   1:  PR[91,2] = PR[90,2] + 22.034;
   1:  PR[91,3] = PR[90,3] + 65.717;
   1:L PR[91] R[100]mm/sec CNT100;
   1:  PR[91,1] = PR[90,1] + 10.623;
   1:  PR[91,2] = PR[90,2] + 22.336;
   1:  PR[91,3] = PR[90,3] + 65.729;
   1:L PR[91] R[100]mm/sec CNT100;
   1:  PR[91,1] = PR[90,1] + 9.950;
   1:  PR[91,2] = PR[90,2] + 22.653;
   1:  PR[91,3] = PR[90,3] + 65.735;
   1:L PR[91] R[100]mm/sec CNT100;
   1:  PR[91,1] = PR[90,1] + 8.633;
   1:  PR[91,2] = PR[90,2] + 23.204;
   1:  PR[91,3] = PR[90,3] + 65.741;
   1:L PR[91] R[100]mm/sec CNT100;
   1:  PR[91,1] = PR[90,1] + 7.929;
   1:  PR[91,2] = PR[90,2] + 23.461;
   1:  PR[91,3] = PR[90,3] + 65.754;
   1:L PR[91] R[100]mm/sec CNT100;
   1:  PR[91,1] = PR[90,1] + 6.878;
   1:  PR[91,2] = PR[90,2] + 23.802;
   1:  PR[91,3] = PR[90,3] + 65.760;
   1:L PR[91] R[100]mm/sec CNT100;
   1:  PR[91,1] = PR[90,1] + 5.935;
   1:  PR[91,2] = PR[90,2] + 24.064;
   1:  PR[91,3] = PR[90,3] + 65.770;
   1:L PR[91] R[100]mm/sec CNT100;
   1:  PR[91,1] = PR[90,1] + 4.733;
   1:  PR[91,2] = PR[90,2] + 24.340;
   1:  PR[91,3] = PR[90,3] + 65.778;
   1:L PR[91] R[100]mm/sec CNT100;
   1:  PR[91,1] = PR[90,1] + 4.119;
   1:  PR[91,2] = PR[90,2] + 24.456;
   1:  PR[91,3] = PR[90,3] + 65.789;
   1:L PR[91] R[100]mm/sec CNT100;
   1:  PR[91,1] = PR[90,1] + 3.151;
   1:  PR[91,2] = PR[90,2] + 24.606;
   1:  PR[91,3] = PR[90,3] + 65.794;
   1:L PR[91] R[100]mm/sec CNT100;
   1:  PR[91,1] = PR[90,1] + 1.922;
   1:  PR[91,2] = PR[90,2] + 24.742;
   1:  PR[91,3] = PR[90,3] + 65.803;
   1:L PR[91] R[100]mm/sec CNT100;
   1:  PR[91,1] = PR[90,1] + 0.859;
   1:  PR[91,2] = PR[90,2] + 24.805;
   1:  PR[91,3] = PR[90,3] + 65.813;
   1:L PR[91] R[100]mm/sec CNT100;
   1:  PR[91,1] = PR[90,1] + -0.123;
   1:  PR[91,2] = PR[90,2] + 24.827;
   1:  PR[91,3] = PR[90,3] + 65.823;
   1:L PR[91] R[100]mm/sec CNT100;
   1:  PR[91,1] = PR[90,1] + -0.555;
   1:  PR[91,2] = PR[90,2] + 24.821;
   1:  PR[91,3] = PR[90,3] + 65.831;
   1:L PR[91] R[100]mm/sec CNT100;
   1:  PR[91,1] = PR[90,1] + -1.536;
   1:  PR[91,2] = PR[90,2] + 24.786;
   1:  PR[91,3] = PR[90,3] + 65.835;
   1:L PR[91] R[100]mm/sec CNT100;
   1:  PR[91,1] = PR[90,1] + -2.957;
   1:  PR[91,2] = PR[90,2] + 24.662;
   1:  PR[91,3] = PR[90,3] + 65.843;
   1:L PR[91] R[100]mm/sec CNT100;
   1:  PR[91,1] = PR[90,1] + -3.734;
   1:  PR[91,2] = PR[90,2] + 24.557;
   1:  PR[91,3] = PR[90,3] + 65.856;
   1:L PR[91] R[100]mm/sec CNT100;
   1:  PR[91,1] = PR[90,1] + -4.789;
   1:  PR[91,2] = PR[90,2] + 24.375;
   1:  PR[91,3] = PR[90,3] + 65.863;
   1:L PR[91] R[100]mm/sec CNT100;
   1:  PR[91,1] = PR[90,1] + -5.745;
   1:  PR[91,2] = PR[90,2] + 24.169;
   1:  PR[91,3] = PR[90,3] + 65.872;
   1:L PR[91] R[100]mm/sec CNT100;
   1:  PR[91,1] = PR[90,1] + -6.960;
   1:  PR[91,2] = PR[90,2] + 23.849;
   1:  PR[91,3] = PR[90,3] + 65.880;
   1:L PR[91] R[100]mm/sec CNT100;
   1:  PR[91,1] = PR[90,1] + -7.532;
   1:  PR[91,2] = PR[90,2] + 23.674;
   1:  PR[91,3] = PR[90,3] + 65.891;
   1:L PR[91] R[100]mm/sec CNT100;
   1:  PR[91,1] = PR[90,1] + -8.875;
   1:  PR[91,2] = PR[90,2] + 23.202;
   1:  PR[91,3] = PR[90,3] + 65.897;
   1:L PR[91] R[100]mm/sec CNT100;
   1:  PR[91,1] = PR[90,1] + -10.185;
   1:  PR[91,2] = PR[90,2] + 22.654;
   1:  PR[91,3] = PR[90,3] + 65.909;
   1:L PR[91] R[100]mm/sec CNT100;
   1:  PR[91,1] = PR[90,1] + -11.460;
   1:  PR[91,2] = PR[90,2] + 22.032;
   1:  PR[91,3] = PR[90,3] + 65.921;
   1:L PR[91] R[100]mm/sec CNT100;
   1:  PR[91,1] = PR[90,1] + -12.697;
   1:  PR[91,2] = PR[90,2] + 21.336;
   1:  PR[91,3] = PR[90,3] + 65.934;
   1:L PR[91] R[100]mm/sec CNT100;
   1:  PR[91,1] = PR[90,1] + -13.891;
   1:  PR[91,2] = PR[90,2] + 20.569;
   1:  PR[91,3] = PR[90,3] + 65.946;
   1:L PR[91] R[100]mm/sec CNT100;
   1:  PR[91,1] = PR[90,1] + -15.043;
   1:  PR[91,2] = PR[90,2] + 19.731;
   1:  PR[91,3] = PR[90,3] + 65.958;
   1:L PR[91] R[100]mm/sec CNT100;
   1:  PR[91,1] = PR[90,1] + -15.381;
   1:  PR[91,2] = PR[90,2] + 19.464;
   1:  PR[91,3] = PR[90,3] + 65.970;
   1:L PR[91] R[100]mm/sec CNT100;
   1:  PR[91,1] = PR[90,1] + -15.929;
   1:  PR[91,2] = PR[90,2] + 19.011;
   1:  PR[91,3] = PR[90,3] + 65.974;
   1:L PR[91] R[100]mm/sec CNT100;
   1:  PR[91,1] = PR[90,1] + -16.463;
   1:  PR[91,2] = PR[90,2] + 18.544;
   1:  PR[91,3] = PR[90,3] + 65.980;
   1:L PR[91] R[100]mm/sec CNT100;
   1:  PR[91,1] = PR[90,1] + -17.190;
   1:  PR[91,2] = PR[90,2] + 17.860;
   1:  PR[91,3] = PR[90,3] + 65.987;
   1:L PR[91] R[100]mm/sec CNT100;
   1:  PR[91,1] = PR[90,1] + -18.206;
   1:  PR[91,2] = PR[90,2] + 16.803;
   1:  PR[91,3] = PR[90,3] + 65.995;
   1:L PR[91] R[100]mm/sec CNT100;
   1:  PR[91,1] = PR[90,1] + -18.610;
   1:  PR[91,2] = PR[90,2] + 16.347;
   1:  PR[91,3] = PR[90,3] + 66.008;
   1:L PR[91] R[100]mm/sec CNT100;
   1:  PR[91,1] = PR[90,1] + -19.433;
   1:  PR[91,2] = PR[90,2] + 15.338;
   1:  PR[91,3] = PR[90,3] + 66.013;
   1:L PR[91] R[100]mm/sec CNT100;
   1:  PR[91,1] = PR[90,1] + -20.289;
   1:  PR[91,2] = PR[90,2] + 14.158;
   1:  PR[91,3] = PR[90,3] + 66.025;
   1:L PR[91] R[100]mm/sec CNT100;
   1:  PR[91,1] = PR[90,1] + -21.075;
   1:  PR[91,2] = PR[90,2] + 12.925;
   1:  PR[91,3] = PR[90,3] + 66.037;
   1:L PR[91] R[100]mm/sec CNT100;
   1:  PR[91,1] = PR[90,1] + -21.521;
   1:  PR[91,2] = PR[90,2] + 12.145;
   1:  PR[91,3] = PR[90,3] + 66.050;
   1:L PR[91] R[100]mm/sec CNT100;
   1:  PR[91,1] = PR[90,1] + -21.781;
   1:  PR[91,2] = PR[90,2] + 11.657;
   1:  PR[91,3] = PR[90,3] + 66.058;
   1:L PR[91] R[100]mm/sec CNT100;
   1:  PR[91,1] = PR[90,1] + -22.223;
   1:  PR[91,2] = PR[90,2] + 10.758;
   1:  PR[91,3] = PR[90,3] + 66.062;
   1:L PR[91] R[100]mm/sec CNT100;
   1:  PR[91,1] = PR[90,1] + -22.593;
   1:  PR[91,2] = PR[90,2] + 9.919;
   1:  PR[91,3] = PR[90,3] + 66.071;
   1:L PR[91] R[100]mm/sec CNT100;
   1:  PR[91,1] = PR[90,1] + -22.966;
   1:  PR[91,2] = PR[90,2] + 8.992;
   1:  PR[91,3] = PR[90,3] + 66.079;
   1:L PR[91] R[100]mm/sec CNT100;
   1:  PR[91,1] = PR[90,1] + -23.437;
   1:  PR[91,2] = PR[90,2] + 7.611;
   1:  PR[91,3] = PR[90,3] + 66.088;
   1:L PR[91] R[100]mm/sec CNT100;
   1:  PR[91,1] = PR[90,1] + -23.825;
   1:  PR[91,2] = PR[90,2] + 6.203;
   1:  PR[91,3] = PR[90,3] + 66.100;
   1:L PR[91] R[100]mm/sec CNT100;
   1:  PR[91,1] = PR[90,1] + -24.040;
   1:  PR[91,2] = PR[90,2] + 5.229;
   1:  PR[91,3] = PR[90,3] + 66.113;
   1:L PR[91] R[100]mm/sec CNT100;
   1:  PR[91,1] = PR[90,1] + -24.202;
   1:  PR[91,2] = PR[90,2] + 4.326;
   1:  PR[91,3] = PR[90,3] + 66.122;
   1:L PR[91] R[100]mm/sec CNT100;
   1:  PR[91,1] = PR[90,1] + -24.344;
   1:  PR[91,2] = PR[90,2] + 3.341;
   1:  PR[91,3] = PR[90,3] + 66.130;
   1:L PR[91] R[100]mm/sec CNT100;
   1:  PR[91,1] = PR[90,1] + -24.475;
   1:  PR[91,2] = PR[90,2] + 1.887;
   1:  PR[91,3] = PR[90,3] + 66.138;
   1:L PR[91] R[100]mm/sec CNT100;
   1:  PR[91,1] = PR[90,1] + -24.519;
   1:  PR[91,2] = PR[90,2] + 0.428;
   1:  PR[91,3] = PR[90,3] + 66.151;
   1:L PR[91] R[100]mm/sec CNT100;
   1:  PR[91,1] = PR[90,1] + -24.475;
   1:  PR[91,2] = PR[90,2] + -1.037;
   1:  PR[91,3] = PR[90,3] + 66.164;
   1:L PR[91] R[100]mm/sec CNT100;
   1:  PR[91,1] = PR[90,1] + -24.442;
   1:  PR[91,2] = PR[90,2] + -1.485;
   1:  PR[91,3] = PR[90,3] + 66.176;
   1:L PR[91] R[100]mm/sec CNT100;
   1:  PR[91,1] = PR[90,1] + -24.345;
   1:  PR[91,2] = PR[90,2] + -2.482;
   1:  PR[91,3] = PR[90,3] + 66.180;
   1:L PR[91] R[100]mm/sec CNT100;
   1:  PR[91,1] = PR[90,1] + -24.128;
   1:  PR[91,2] = PR[90,2] + -3.923;
   1:  PR[91,3] = PR[90,3] + 66.189;
   1:L PR[91] R[100]mm/sec CNT100;
   1:  PR[91,1] = PR[90,1] + -23.825;
   1:  PR[91,2] = PR[90,2] + -5.351;
   1:  PR[91,3] = PR[90,3] + 66.202;
   1:L PR[91] R[100]mm/sec CNT100;
   1:  PR[91,1] = PR[90,1] + -23.581;
   1:  PR[91,2] = PR[90,2] + -6.240;
   1:  PR[91,3] = PR[90,3] + 66.214;
   1:L PR[91] R[100]mm/sec CNT100;
   1:  PR[91,1] = PR[90,1] + -23.438;
   1:  PR[91,2] = PR[90,2] + -6.755;
   1:  PR[91,3] = PR[90,3] + 66.222;
   1:L PR[91] R[100]mm/sec CNT100;
   1:  PR[91,1] = PR[90,1] + -22.967;
   1:  PR[91,2] = PR[90,2] + -8.135;
   1:  PR[91,3] = PR[90,3] + 66.227;
   1:L PR[91] R[100]mm/sec CNT100;
   1:  PR[91,1] = PR[90,1] + -22.414;
   1:  PR[91,2] = PR[90,2] + -9.486;
   1:  PR[91,3] = PR[90,3] + 66.240;
   1:L PR[91] R[100]mm/sec CNT100;
   1:  PR[91,1] = PR[90,1] + -21.780;
   1:  PR[91,2] = PR[90,2] + -10.804;
   1:  PR[91,3] = PR[90,3] + 66.252;
   1:L PR[91] R[100]mm/sec CNT100;
   1:  PR[91,1] = PR[90,1] + -21.521;
   1:  PR[91,2] = PR[90,2] + -11.289;
   1:  PR[91,3] = PR[90,3] + 66.265;
   1:L PR[91] R[100]mm/sec CNT100;
   1:  PR[91,1] = PR[90,1] + -21.075;
   1:  PR[91,2] = PR[90,2] + -12.070;
   1:  PR[91,3] = PR[90,3] + 66.270;
   1:L PR[91] R[100]mm/sec CNT100;
   1:  PR[91,1] = PR[90,1] + -20.289;
   1:  PR[91,2] = PR[90,2] + -13.303;
   1:  PR[91,3] = PR[90,3] + 66.278;
   1:L PR[91] R[100]mm/sec CNT100;
   1:  PR[91,1] = PR[90,1] + -19.431;
   1:  PR[91,2] = PR[90,2] + -14.485;
   1:  PR[91,3] = PR[90,3] + 66.290;
   1:L PR[91] R[100]mm/sec CNT100;
   1:  PR[91,1] = PR[90,1] + -18.908;
   1:  PR[91,2] = PR[90,2] + -15.137;
   1:  PR[91,3] = PR[90,3] + 66.303;
   1:L PR[91] R[100]mm/sec CNT100;
   1:  PR[91,1] = PR[90,1] + -18.204;
   1:  PR[91,2] = PR[90,2] + -15.950;
   1:  PR[91,3] = PR[90,3] + 66.310;
   1:L PR[91] R[100]mm/sec CNT100;
   1:  PR[91,1] = PR[90,1] + -17.190;
   1:  PR[91,2] = PR[90,2] + -17.005;
   1:  PR[91,3] = PR[90,3] + 66.319;
   1:L PR[91] R[100]mm/sec CNT100;
   1:  PR[91,1] = PR[90,1] + -16.465;
   1:  PR[91,2] = PR[90,2] + -17.687;
   1:  PR[91,3] = PR[90,3] + 66.332;
   1:L PR[91] R[100]mm/sec CNT100;
   1:  PR[91,1] = PR[90,1] + -15.590;
   1:  PR[91,2] = PR[90,2] + -18.440;
   1:  PR[91,3] = PR[90,3] + 66.341;
   1:L PR[91] R[100]mm/sec CNT100;
   1:  PR[91,1] = PR[90,1] + -15.042;
   1:  PR[91,2] = PR[90,2] + -18.877;
   1:  PR[91,3] = PR[90,3] + 66.351;
   1:L PR[91] R[100]mm/sec CNT100;
   1:  PR[91,1] = PR[90,1] + -13.891;
   1:  PR[91,2] = PR[90,2] + -19.714;
   1:  PR[91,3] = PR[90,3] + 66.357;
   1:L PR[91] R[100]mm/sec CNT100;
   1:  PR[91,1] = PR[90,1] + -12.718;
   1:  PR[91,2] = PR[90,2] + -20.468;
   1:  PR[91,3] = PR[90,3] + 66.369;
   1:L PR[91] R[100]mm/sec CNT100;
   1:  PR[91,1] = PR[90,1] + -11.460;
   1:  PR[91,2] = PR[90,2] + -21.177;
   1:  PR[91,3] = PR[90,3] + 66.381;
   1:L PR[91] R[100]mm/sec CNT100;
   1:  PR[91,1] = PR[90,1] + -10.185;
   1:  PR[91,2] = PR[90,2] + -21.799;
   1:  PR[91,3] = PR[90,3] + 66.394;
   1:L PR[91] R[100]mm/sec CNT100;
   1:  PR[91,1] = PR[90,1] + -8.875;
   1:  PR[91,2] = PR[90,2] + -22.347;
   1:  PR[91,3] = PR[90,3] + 66.406;
   1:L PR[91] R[100]mm/sec CNT100;
   1:  PR[91,1] = PR[90,1] + -7.532;
   1:  PR[91,2] = PR[90,2] + -22.819;
   1:  PR[91,3] = PR[90,3] + 66.418;
   1:L PR[91] R[100]mm/sec CNT100;
   1:  PR[91,1] = PR[90,1] + -6.960;
   1:  PR[91,2] = PR[90,2] + -22.994;
   1:  PR[91,3] = PR[90,3] + 66.431;
   1:L PR[91] R[100]mm/sec CNT100;
   1:  PR[91,1] = PR[90,1] + -5.748;
   1:  PR[91,2] = PR[90,2] + -23.313;
   1:  PR[91,3] = PR[90,3] + 66.436;
   1:L PR[91] R[100]mm/sec CNT100;
   1:  PR[91,1] = PR[90,1] + -4.356;
   1:  PR[91,2] = PR[90,2] + -23.601;
   1:  PR[91,3] = PR[90,3] + 66.447;
   1:L PR[91] R[100]mm/sec CNT100;
   1:  PR[91,1] = PR[90,1] + -2.951;
   1:  PR[91,2] = PR[90,2] + -23.807;
   1:  PR[91,3] = PR[90,3] + 66.459;
   1:L PR[91] R[100]mm/sec CNT100;
   1:  PR[91,1] = PR[90,1] + -1.977;
   1:  PR[91,2] = PR[90,2] + -23.900;
   1:  PR[91,3] = PR[90,3] + 66.472;
   1:L PR[91] R[100]mm/sec CNT100;
   1:  PR[91,1] = PR[90,1] + -0.911;
   1:  PR[91,2] = PR[90,2] + -23.959;
   1:  PR[91,3] = PR[90,3] + 66.480;
   1:L PR[91] R[100]mm/sec CNT100;
   1:  PR[91,1] = PR[90,1] + 0.321;
   1:  PR[91,2] = PR[90,2] + -23.966;
   1:  PR[91,3] = PR[90,3] + 66.489;
   1:L PR[91] R[100]mm/sec CNT100;
   1:  PR[91] = PR[90];
   1:  PR[91,1] = PR[90,1] + 1.327;
   1:  PR[91,2] = PR[90,2] + -23.929;
   1:  PR[91,3] = PR[90,3] + 67.830;
   1:L PR[91] R[100]mm/sec CNT100;
   1:  PR[91,1] = PR[90,1] + 1.891;
   1:  PR[91,2] = PR[90,2] + -23.889;
   1:  PR[91,3] = PR[90,3] + 66.513;
   1:L PR[91] R[100]mm/sec CNT100;
   1:  PR[91,1] = PR[90,1] + 3.010;
   1:  PR[91,2] = PR[90,2] + -23.769;
   1:  PR[91,3] = PR[90,3] + 66.517;
   1:L PR[91] R[100]mm/sec CNT100;
   1:  PR[91,1] = PR[90,1] + 4.436;
   1:  PR[91,2] = PR[90,2] + -23.542;
   1:  PR[91,3] = PR[90,3] + 66.527;
   1:L PR[91] R[100]mm/sec CNT100;
   1:  PR[91,1] = PR[90,1] + 5.595;
   1:  PR[91,2] = PR[90,2] + -23.293;
   1:  PR[91,3] = PR[90,3] + 66.540;
   1:L PR[91] R[100]mm/sec CNT100;
   1:  PR[91,1] = PR[90,1] + 6.992;
   1:  PR[91,2] = PR[90,2] + -22.912;
   1:  PR[91,3] = PR[90,3] + 66.550;
   1:L PR[91] R[100]mm/sec CNT100;
   1:  PR[91,1] = PR[90,1] + 7.839;
   1:  PR[91,2] = PR[90,2] + -22.637;
   1:  PR[91,3] = PR[90,3] + 66.563;
   1:L PR[91] R[100]mm/sec CNT100;
   1:  PR[91,1] = PR[90,1] + 8.828;
   1:  PR[91,2] = PR[90,2] + -22.269;
   1:  PR[91,3] = PR[90,3] + 66.570;
   1:L PR[91] R[100]mm/sec CNT100;
   1:  PR[91,1] = PR[90,1] + 9.928;
   1:  PR[91,2] = PR[90,2] + -21.807;
   1:  PR[91,3] = PR[90,3] + 66.580;
   1:L PR[91] R[100]mm/sec CNT100;
   1:  PR[91,1] = PR[90,1] + 10.637;
   1:  PR[91,2] = PR[90,2] + -21.474;
   1:  PR[91,3] = PR[90,3] + 66.590;
   1:L PR[91] R[100]mm/sec CNT100;
   1:  PR[91,1] = PR[90,1] + 11.216;
   1:  PR[91,2] = PR[90,2] + -21.180;
   1:  PR[91,3] = PR[90,3] + 66.597;
   1:L PR[91] R[100]mm/sec CNT100;
   1:  PR[91,1] = PR[90,1] + 12.479;
   1:  PR[91,2] = PR[90,2] + -20.468;
   1:  PR[91,3] = PR[90,3] + 66.602;
   1:L PR[91] R[100]mm/sec CNT100;
   1:  PR[91,1] = PR[90,1] + 13.379;
   1:  PR[91,2] = PR[90,2] + -19.896;
   1:  PR[91,3] = PR[90,3] + 66.615;
   1:L PR[91] R[100]mm/sec CNT100;
   1:  PR[91,1] = PR[90,1] + 13.896;
   1:  PR[91,2] = PR[90,2] + -19.544;
   1:  PR[91,3] = PR[90,3] + 66.624;
   1:L PR[91] R[100]mm/sec CNT100;
   1:  PR[91,1] = PR[90,1] + 15.053;
   1:  PR[91,2] = PR[90,2] + -18.680;
   1:  PR[91,3] = PR[90,3] + 66.630;
   1:L PR[91] R[100]mm/sec CNT100;
   1:  PR[91,1] = PR[90,1] + 16.161;
   1:  PR[91,2] = PR[90,2] + -17.746;
   1:  PR[91,3] = PR[90,3] + 66.642;
   1:L PR[91] R[100]mm/sec CNT100;
   1:  PR[91,1] = PR[90,1] + 16.640;
   1:  PR[91,2] = PR[90,2] + -17.305;
   1:  PR[91,3] = PR[90,3] + 66.655;
   1:L PR[91] R[100]mm/sec CNT100;
   1:  PR[91,1] = PR[90,1] + 17.215;
   1:  PR[91,2] = PR[90,2] + -16.743;
   1:  PR[91,3] = PR[90,3] + 66.660;
   1:L PR[91] R[100]mm/sec CNT100;
   1:  PR[91,1] = PR[90,1] + 18.217;
   1:  PR[91,2] = PR[90,2] + -15.669;
   1:  PR[91,3] = PR[90,3] + 66.667;
   1:L PR[91] R[100]mm/sec CNT100;
   1:  PR[91,1] = PR[90,1] + 18.987;
   1:  PR[91,2] = PR[90,2] + -14.747;
   1:  PR[91,3] = PR[90,3] + 66.680;
   1:L PR[91] R[100]mm/sec CNT100;
   1:  PR[91,1] = PR[90,1] + 19.539;
   1:  PR[91,2] = PR[90,2] + -14.025;
   1:  PR[91,3] = PR[90,3] + 66.690;
   1:L PR[91] R[100]mm/sec CNT100;
   1:  PR[91,1] = PR[90,1] + 20.011;
   1:  PR[91,2] = PR[90,2] + -13.361;
   1:  PR[91,3] = PR[90,3] + 66.698;
   1:L PR[91] R[100]mm/sec CNT100;
   1:  PR[91,1] = PR[90,1] + 20.805;
   1:  PR[91,2] = PR[90,2] + -12.123;
   1:  PR[91,3] = PR[90,3] + 66.705;
   1:L PR[91] R[100]mm/sec CNT100;
   1:  PR[91,1] = PR[90,1] + 21.394;
   1:  PR[91,2] = PR[90,2] + -11.082;
   1:  PR[91,3] = PR[90,3] + 66.718;
   1:L PR[91] R[100]mm/sec CNT100;
   1:  PR[91,1] = PR[90,1] + 22.047;
   1:  PR[91,2] = PR[90,2] + -9.767;
   1:  PR[91,3] = PR[90,3] + 66.729;
   1:L PR[91] R[100]mm/sec CNT100;
   1:  PR[91,1] = PR[90,1] + 22.421;
   1:  PR[91,2] = PR[90,2] + -8.915;
   1:  PR[91,3] = PR[90,3] + 66.741;
   1:L PR[91] R[100]mm/sec CNT100;
   1:  PR[91,1] = PR[90,1] + 22.713;
   1:  PR[91,2] = PR[90,2] + -8.176;
   1:  PR[91,3] = PR[90,3] + 66.749;
   1:L PR[91] R[100]mm/sec CNT100;
   1:  PR[91,1] = PR[90,1] + 23.189;
   1:  PR[91,2] = PR[90,2] + -6.788;
   1:  PR[91,3] = PR[90,3] + 66.756;
   1:L PR[91] R[100]mm/sec CNT100;
   1:  PR[91,1] = PR[90,1] + 23.580;
   1:  PR[91,2] = PR[90,2] + -5.375;
   1:  PR[91,3] = PR[90,3] + 66.769;
   1:L PR[91] R[100]mm/sec CNT100;
   1:  PR[91,1] = PR[90,1] + 23.836;
   1:  PR[91,2] = PR[90,2] + -4.201;
   1:  PR[91,3] = PR[90,3] + 66.782;
   1:L PR[91] R[100]mm/sec CNT100;
   1:  PR[91,1] = PR[90,1] + 23.929;
   1:  PR[91,2] = PR[90,2] + -3.684;
   1:  PR[91,3] = PR[90,3] + 66.792;
   1:L PR[91] R[100]mm/sec CNT100;
   1:  PR[91,1] = PR[90,1] + 24.105;
   1:  PR[91,2] = PR[90,2] + -2.497;
   1:  PR[91,3] = PR[90,3] + 66.797;
   1:L PR[91] R[100]mm/sec CNT100;
   1:  PR[91,1] = PR[90,1] + 24.217;
   1:  PR[91,2] = PR[90,2] + -1.302;
   1:  PR[91,3] = PR[90,3] + 66.807;
   1:L PR[91] R[100]mm/sec CNT100;
   1:  PR[91,1] = PR[90,1] + 24.248;
   1:  PR[91,2] = PR[90,2] + -0.778;
   1:  PR[91,3] = PR[90,3] + 66.818;
   1:L PR[91] R[100]mm/sec CNT100;
   1:  PR[91,1] = PR[90,1] + 24.281;
   1:  PR[91,2] = PR[90,2] + 0.427;
   1:  PR[91,3] = PR[90,3] + 66.822;
   1:L PR[91] R[100]mm/sec CNT100;
   1:  PR[91,1] = PR[90,1] + 24.236;
   1:  PR[91,2] = PR[90,2] + 1.895;
   1:  PR[91,3] = PR[90,3] + 66.833;
   1:L PR[91] R[100]mm/sec CNT100;
   1:  PR[91,1] = PR[90,1] + 24.104;
   1:  PR[91,2] = PR[90,2] + 3.353;
   1:  PR[91,3] = PR[90,3] + 66.845;
   1:L PR[91] R[100]mm/sec CNT100;
   1:  PR[91,1] = PR[90,1] + 23.886;
   1:  PR[91,2] = PR[90,2] + 4.796;
   1:  PR[91,3] = PR[90,3] + 66.858;
   1:L PR[91] R[100]mm/sec CNT100;
   1:  PR[91,1] = PR[90,1] + 23.513;
   1:  PR[91,2] = PR[90,2] + 6.492;
   1:  PR[91,3] = PR[90,3] + 66.871;
   1:L PR[91] R[100]mm/sec CNT100;
   1:  PR[91,1] = PR[90,1] + 23.189;
   1:  PR[91,2] = PR[90,2] + 7.642;
   1:  PR[91,3] = PR[90,3] + 66.886;
   1:L PR[91] R[100]mm/sec CNT100;
   1:  PR[91,1] = PR[90,1] + 22.713;
   1:  PR[91,2] = PR[90,2] + 9.031;
   1:  PR[91,3] = PR[90,3] + 66.896;
   1:L PR[91] R[100]mm/sec CNT100;
   1:  PR[91,1] = PR[90,1] + 22.421;
   1:  PR[91,2] = PR[90,2] + 9.770;
   1:  PR[91,3] = PR[90,3] + 66.909;
   1:L PR[91] R[100]mm/sec CNT100;
   1:  PR[91,1] = PR[90,1] + 22.046;
   1:  PR[91,2] = PR[90,2] + 10.624;
   1:  PR[91,3] = PR[90,3] + 66.916;
   1:L PR[91] R[100]mm/sec CNT100;
   1:  PR[91,1] = PR[90,1] + 21.520;
   1:  PR[91,2] = PR[90,2] + 11.700;
   1:  PR[91,3] = PR[90,3] + 66.924;
   1:L PR[91] R[100]mm/sec CNT100;
   1:  PR[91,1] = PR[90,1] + 20.804;
   1:  PR[91,2] = PR[90,2] + 12.979;
   1:  PR[91,3] = PR[90,3] + 66.934;
   1:L PR[91] R[100]mm/sec CNT100;
   1:  PR[91,1] = PR[90,1] + 20.011;
   1:  PR[91,2] = PR[90,2] + 14.215;
   1:  PR[91,3] = PR[90,3] + 66.947;
   1:L PR[91] R[100]mm/sec CNT100;
   1:  PR[91,1] = PR[90,1] + 19.378;
   1:  PR[91,2] = PR[90,2] + 15.097;
   1:  PR[91,3] = PR[90,3] + 66.960;
   1:L PR[91] R[100]mm/sec CNT100;
   1:  PR[91,1] = PR[90,1] + 18.989;
   1:  PR[91,2] = PR[90,2] + 15.599;
   1:  PR[91,3] = PR[90,3] + 66.969;
   1:L PR[91] R[100]mm/sec CNT100;
   1:  PR[91,1] = PR[90,1] + 18.038;
   1:  PR[91,2] = PR[90,2] + 16.725;
   1:  PR[91,3] = PR[90,3] + 66.975;
   1:L PR[91] R[100]mm/sec CNT100;
   1:  PR[91,1] = PR[90,1] + 17.216;
   1:  PR[91,2] = PR[90,2] + 17.597;
   1:  PR[91,3] = PR[90,3] + 66.987;
   1:L PR[91] R[100]mm/sec CNT100;
   1:  PR[91,1] = PR[90,1] + 16.640;
   1:  PR[91,2] = PR[90,2] + 18.160;
   1:  PR[91,3] = PR[90,3] + 66.998;
   1:L PR[91] R[100]mm/sec CNT100;
   1:  PR[91,1] = PR[90,1] + 16.160;
   1:  PR[91,2] = PR[90,2] + 18.601;
   1:  PR[91,3] = PR[90,3] + 67.005;
   1:L PR[91] R[100]mm/sec CNT100;
   1:  PR[91,1] = PR[90,1] + 15.050;
   1:  PR[91,2] = PR[90,2] + 19.537;
   1:  PR[91,3] = PR[90,3] + 67.010;
   1:L PR[91] R[100]mm/sec CNT100;
   1:  PR[91,1] = PR[90,1] + 14.654;
   1:  PR[91,2] = PR[90,2] + 19.841;
   1:  PR[91,3] = PR[90,3] + 67.023;
   1:L PR[91] R[100]mm/sec CNT100;
   1:  PR[91,1] = PR[90,1] + 13.589;
   1:  PR[91,2] = PR[90,2] + 20.613;
   1:  PR[91,3] = PR[90,3] + 67.027;
   1:L PR[91] R[100]mm/sec CNT100;
   1:  PR[91,1] = PR[90,1] + 12.478;
   1:  PR[91,2] = PR[90,2] + 21.324;
   1:  PR[91,3] = PR[90,3] + 67.039;
   1:L PR[91] R[100]mm/sec CNT100;
   1:  PR[91,1] = PR[90,1] + 11.216;
   1:  PR[91,2] = PR[90,2] + 22.035;
   1:  PR[91,3] = PR[90,3] + 67.050;
   1:L PR[91] R[100]mm/sec CNT100;
   1:  PR[91,1] = PR[90,1] + 10.637;
   1:  PR[91,2] = PR[90,2] + 22.329;
   1:  PR[91,3] = PR[90,3] + 67.063;
   1:L PR[91] R[100]mm/sec CNT100;
   1:  PR[91,1] = PR[90,1] + 9.929;
   1:  PR[91,2] = PR[90,2] + 22.662;
   1:  PR[91,3] = PR[90,3] + 67.068;
   1:L PR[91] R[100]mm/sec CNT100;
   1:  PR[91,1] = PR[90,1] + 8.589;
   1:  PR[91,2] = PR[90,2] + 23.220;
   1:  PR[91,3] = PR[90,3] + 67.075;
   1:L PR[91] R[100]mm/sec CNT100;
   1:  PR[91,1] = PR[90,1] + 7.841;
   1:  PR[91,2] = PR[90,2] + 23.492;
   1:  PR[91,3] = PR[90,3] + 67.088;
   1:L PR[91] R[100]mm/sec CNT100;
   1:  PR[91,1] = PR[90,1] + 6.992;
   1:  PR[91,2] = PR[90,2] + 23.767;
   1:  PR[91,3] = PR[90,3] + 67.095;
   1:L PR[91] R[100]mm/sec CNT100;
   1:  PR[91,1] = PR[90,1] + 5.593;
   1:  PR[91,2] = PR[90,2] + 24.148;
   1:  PR[91,3] = PR[90,3] + 67.102;
   1:L PR[91] R[100]mm/sec CNT100;
   1:  PR[91,1] = PR[90,1] + 4.756;
   1:  PR[91,2] = PR[90,2] + 24.335;
   1:  PR[91,3] = PR[90,3] + 67.115;
   1:L PR[91] R[100]mm/sec CNT100;
   1:  PR[91,1] = PR[90,1] + 4.189;
   1:  PR[91,2] = PR[90,2] + 24.444;
   1:  PR[91,3] = PR[90,3] + 67.122;
   1:L PR[91] R[100]mm/sec CNT100;
   1:  PR[91,1] = PR[90,1] + 3.012;
   1:  PR[91,2] = PR[90,2] + 24.624;
   1:  PR[91,3] = PR[90,3] + 67.127;
   1:L PR[91] R[100]mm/sec CNT100;
   1:  PR[91,1] = PR[90,1] + 1.894;
   1:  PR[91,2] = PR[90,2] + 24.744;
   1:  PR[91,3] = PR[90,3] + 67.138;
   1:L PR[91] R[100]mm/sec CNT100;
   1:  PR[91,1] = PR[90,1] + 1.069;
   1:  PR[91,2] = PR[90,2] + 24.795;
   1:  PR[91,3] = PR[90,3] + 67.148;
   1:L PR[91] R[100]mm/sec CNT100;
   1:  PR[91,1] = PR[90,1] + -0.122;
   1:  PR[91,2] = PR[90,2] + 24.827;
   1:  PR[91,3] = PR[90,3] + 67.155;
   1:L PR[91] R[100]mm/sec CNT100;
   1:  PR[91,1] = PR[90,1] + -0.980;
   1:  PR[91,2] = PR[90,2] + 24.812;
   1:  PR[91,3] = PR[90,3] + 67.165;
   1:L PR[91] R[100]mm/sec CNT100;
   1:  PR[91,1] = PR[90,1] + -1.556;
   1:  PR[91,2] = PR[90,2] + 24.785;
   1:  PR[91,3] = PR[90,3] + 67.173;
   1:L PR[91] R[100]mm/sec CNT100;
   1:  PR[91,1] = PR[90,1] + -3.002;
   1:  PR[91,2] = PR[90,2] + 24.656;
   1:  PR[91,3] = PR[90,3] + 67.178;
   1:L PR[91] R[100]mm/sec CNT100;
   1:  PR[91,1] = PR[90,1] + -3.850;
   1:  PR[91,2] = PR[90,2] + 24.540;
   1:  PR[91,3] = PR[90,3] + 67.190;
   1:L PR[91] R[100]mm/sec CNT100;
   1:  PR[91,1] = PR[90,1] + -4.670;
   1:  PR[91,2] = PR[90,2] + 24.398;
   1:  PR[91,3] = PR[90,3] + 67.198;
   1:L PR[91] R[100]mm/sec CNT100;
   1:  PR[91,1] = PR[90,1] + -6.086;
   1:  PR[91,2] = PR[90,2] + 24.086;
   1:  PR[91,3] = PR[90,3] + 67.205;
   1:L PR[91] R[100]mm/sec CNT100;
   1:  PR[91,1] = PR[90,1] + -6.952;
   1:  PR[91,2] = PR[90,2] + 23.851;
   1:  PR[91,3] = PR[90,3] + 67.217;
   1:L PR[91] R[100]mm/sec CNT100;
   1:  PR[91,1] = PR[90,1] + -7.465;
   1:  PR[91,2] = PR[90,2] + 23.695;
   1:  PR[91,3] = PR[90,3] + 67.225;
   1:L PR[91] R[100]mm/sec CNT100;
   1:  PR[91,1] = PR[90,1] + -8.831;
   1:  PR[91,2] = PR[90,2] + 23.219;
   1:  PR[91,3] = PR[90,3] + 67.230;
   1:L PR[91] R[100]mm/sec CNT100;
   1:  PR[91,1] = PR[90,1] + -10.165;
   1:  PR[91,2] = PR[90,2] + 22.663;
   1:  PR[91,3] = PR[90,3] + 67.242;
   1:L PR[91] R[100]mm/sec CNT100;
   1:  PR[91,1] = PR[90,1] + -11.235;
   1:  PR[91,2] = PR[90,2] + 22.146;
   1:  PR[91,3] = PR[90,3] + 67.255;
   1:L PR[91] R[100]mm/sec CNT100;
   1:  PR[91,1] = PR[90,1] + -11.678;
   1:  PR[91,2] = PR[90,2] + 21.913;
   1:  PR[91,3] = PR[90,3] + 67.265;
   1:L PR[91] R[100]mm/sec CNT100;
   1:  PR[91,1] = PR[90,1] + -12.971;
   1:  PR[91,2] = PR[90,2] + 21.167;
   1:  PR[91,3] = PR[90,3] + 67.270;
   1:L PR[91] R[100]mm/sec CNT100;
   1:  PR[91,1] = PR[90,1] + -13.928;
   1:  PR[91,2] = PR[90,2] + 20.544;
   1:  PR[91,3] = PR[90,3] + 67.282;
   1:L PR[91] R[100]mm/sec CNT100;
   1:  PR[91,1] = PR[90,1] + -15.095;
   1:  PR[91,2] = PR[90,2] + 19.690;
   1:  PR[91,3] = PR[90,3] + 67.292;
   1:L PR[91] R[100]mm/sec CNT100;
   1:  PR[91,1] = PR[90,1] + -15.652;
   1:  PR[91,2] = PR[90,2] + 19.244;
   1:  PR[91,3] = PR[90,3] + 67.305;
   1:L PR[91] R[100]mm/sec CNT100;
   1:  PR[91,1] = PR[90,1] + -16.201;
   1:  PR[91,2] = PR[90,2] + 18.776;
   1:  PR[91,3] = PR[90,3] + 67.311;
   1:L PR[91] R[100]mm/sec CNT100;
   1:  PR[91,1] = PR[90,1] + -17.267;
   1:  PR[91,2] = PR[90,2] + 17.785;
   1:  PR[91,3] = PR[90,3] + 67.317;
   1:L PR[91] R[100]mm/sec CNT100;
   1:  PR[91,1] = PR[90,1] + -18.456;
   1:  PR[91,2] = PR[90,2] + 16.524;
   1:  PR[91,3] = PR[90,3] + 67.330;
   1:L PR[91] R[100]mm/sec CNT100;
   1:  PR[91,1] = PR[90,1] + -19.390;
   1:  PR[91,2] = PR[90,2] + 15.393;
   1:  PR[91,3] = PR[90,3] + 67.345;
   1:L PR[91] R[100]mm/sec CNT100;
   1:  PR[91,1] = PR[90,1] + -20.097;
   1:  PR[91,2] = PR[90,2] + 14.434;
   1:  PR[91,3] = PR[90,3] + 67.358;
   1:L PR[91] R[100]mm/sec CNT100;
   1:  PR[91,1] = PR[90,1] + -21.043;
   1:  PR[91,2] = PR[90,2] + 12.978;
   1:  PR[91,3] = PR[90,3] + 67.368;
   1:L PR[91] R[100]mm/sec CNT100;
   1:  PR[91,1] = PR[90,1] + -21.759;
   1:  PR[91,2] = PR[90,2] + 11.700;
   1:  PR[91,3] = PR[90,3] + 67.383;
   1:L PR[91] R[100]mm/sec CNT100;
   1:  PR[91,1] = PR[90,1] + -22.283;
   1:  PR[91,2] = PR[90,2] + 10.627;
   1:  PR[91,3] = PR[90,3] + 67.396;
   1:L PR[91] R[100]mm/sec CNT100;
   1:  PR[91,1] = PR[90,1] + -22.858;
   1:  PR[91,2] = PR[90,2] + 9.271;
   1:  PR[91,3] = PR[90,3] + 67.406;
   1:L PR[91] R[100]mm/sec CNT100;
   1:  PR[91,1] = PR[90,1] + -23.040;
   1:  PR[91,2] = PR[90,2] + 8.781;
   1:  PR[91,3] = PR[90,3] + 67.419;
   1:L PR[91] R[100]mm/sec CNT100;
   1:  PR[91,1] = PR[90,1] + -23.427;
   1:  PR[91,2] = PR[90,2] + 7.644;
   1:  PR[91,3] = PR[90,3] + 67.424;
   1:L PR[91] R[100]mm/sec CNT100;
   1:  PR[91,1] = PR[90,1] + -23.818;
   1:  PR[91,2] = PR[90,2] + 6.231;
   1:  PR[91,3] = PR[90,3] + 67.434;
   1:L PR[91] R[100]mm/sec CNT100;
   1:  PR[91,1] = PR[90,1] + -24.125;
   1:  PR[91,2] = PR[90,2] + 4.797;
   1:  PR[91,3] = PR[90,3] + 67.447;
   1:L PR[91] R[100]mm/sec CNT100;
   1:  PR[91,1] = PR[90,1] + -24.307;
   1:  PR[91,2] = PR[90,2] + 3.618;
   1:  PR[91,3] = PR[90,3] + 67.459;
   1:L PR[91] R[100]mm/sec CNT100;
   1:  PR[91,1] = PR[90,1] + -24.455;
   1:  PR[91,2] = PR[90,2] + 2.155;
   1:  PR[91,3] = PR[90,3] + 67.470;
   1:L PR[91] R[100]mm/sec CNT100;
   1:  PR[91,1] = PR[90,1] + -24.486;
   1:  PR[91,2] = PR[90,2] + 1.634;
   1:  PR[91,3] = PR[90,3] + 67.483;
   1:L PR[91] R[100]mm/sec CNT100;
   1:  PR[91,1] = PR[90,1] + -24.519;
   1:  PR[91,2] = PR[90,2] + 0.428;
   1:  PR[91,3] = PR[90,3] + 67.487;
   1:L PR[91] R[100]mm/sec CNT100;
   1:  PR[91,1] = PR[90,1] + -24.474;
   1:  PR[91,2] = PR[90,2] + -1.040;
   1:  PR[91,3] = PR[90,3] + 67.498;
   1:L PR[91] R[100]mm/sec CNT100;
   1:  PR[91,1] = PR[90,1] + -24.343;
   1:  PR[91,2] = PR[90,2] + -2.498;
   1:  PR[91,3] = PR[90,3] + 67.510;
   1:L PR[91] R[100]mm/sec CNT100;
   1:  PR[91,1] = PR[90,1] + -24.124;
   1:  PR[91,2] = PR[90,2] + -3.943;
   1:  PR[91,3] = PR[90,3] + 67.523;
   1:L PR[91] R[100]mm/sec CNT100;
   1:  PR[91,1] = PR[90,1] + -23.818;
   1:  PR[91,2] = PR[90,2] + -5.377;
   1:  PR[91,3] = PR[90,3] + 67.536;
   1:L PR[91] R[100]mm/sec CNT100;
   1:  PR[91,1] = PR[90,1] + -23.679;
   1:  PR[91,2] = PR[90,2] + -5.885;
   1:  PR[91,3] = PR[90,3] + 67.548;
   1:L PR[91] R[100]mm/sec CNT100;
   1:  PR[91,1] = PR[90,1] + -23.428;
   1:  PR[91,2] = PR[90,2] + -6.788;
   1:  PR[91,3] = PR[90,3] + 67.553;
   1:L PR[91] R[100]mm/sec CNT100;
   1:  PR[91,1] = PR[90,1] + -22.953;
   1:  PR[91,2] = PR[90,2] + -8.172;
   1:  PR[91,3] = PR[90,3] + 67.561;
   1:L PR[91] R[100]mm/sec CNT100;
   1:  PR[91,1] = PR[90,1] + -22.395;
   1:  PR[91,2] = PR[90,2] + -9.528;
   1:  PR[91,3] = PR[90,3] + 67.574;
   1:L PR[91] R[100]mm/sec CNT100;
   1:  PR[91,1] = PR[90,1] + -21.755;
   1:  PR[91,2] = PR[90,2] + -10.852;
   1:  PR[91,3] = PR[90,3] + 67.587;
   1:L PR[91] R[100]mm/sec CNT100;
   1:  PR[91,1] = PR[90,1] + -21.554;
   1:  PR[91,2] = PR[90,2] + -11.229;
   1:  PR[91,3] = PR[90,3] + 67.599;
   1:L PR[91] R[100]mm/sec CNT100;
   1:  PR[91,1] = PR[90,1] + -21.044;
   1:  PR[91,2] = PR[90,2] + -12.122;
   1:  PR[91,3] = PR[90,3] + 67.603;
   1:L PR[91] R[100]mm/sec CNT100;
   1:  PR[91,1] = PR[90,1] + -20.251;
   1:  PR[91,2] = PR[90,2] + -13.358;
   1:  PR[91,3] = PR[90,3] + 67.612;
   1:L PR[91] R[100]mm/sec CNT100;
   1:  PR[91,1] = PR[90,1] + -19.387;
   1:  PR[91,2] = PR[90,2] + -14.542;
   1:  PR[91,3] = PR[90,3] + 67.625;
   1:L PR[91] R[100]mm/sec CNT100;
   1:  PR[91,1] = PR[90,1] + -18.806;
   1:  PR[91,2] = PR[90,2] + -15.259;
   1:  PR[91,3] = PR[90,3] + 67.637;
   1:L PR[91] R[100]mm/sec CNT100;
   1:  PR[91,1] = PR[90,1] + -18.280;
   1:  PR[91,2] = PR[90,2] + -15.866;
   1:  PR[91,3] = PR[90,3] + 67.645;
   1:L PR[91] R[100]mm/sec CNT100;
   1:  PR[91,1] = PR[90,1] + -17.268;
   1:  PR[91,2] = PR[90,2] + -16.928;
   1:  PR[91,3] = PR[90,3] + 67.652;
   1:L PR[91] R[100]mm/sec CNT100;
   1:  PR[91,1] = PR[90,1] + -16.203;
   1:  PR[91,2] = PR[90,2] + -17.919;
   1:  PR[91,3] = PR[90,3] + 67.665;
   1:L PR[91] R[100]mm/sec CNT100;
   1:  PR[91,1] = PR[90,1] + -15.293;
   1:  PR[91,2] = PR[90,2] + -18.679;
   1:  PR[91,3] = PR[90,3] + 67.678;
   1:L PR[91] R[100]mm/sec CNT100;
   1:  PR[91,1] = PR[90,1] + -14.134;
   1:  PR[91,2] = PR[90,2] + -19.544;
   1:  PR[91,3] = PR[90,3] + 67.688;
   1:L PR[91] R[100]mm/sec CNT100;
   1:  PR[91,1] = PR[90,1] + -13.720;
   1:  PR[91,2] = PR[90,2] + -19.826;
   1:  PR[91,3] = PR[90,3] + 67.701;
   1:L PR[91] R[100]mm/sec CNT100;
   1:  PR[91,1] = PR[90,1] + -12.753;
   1:  PR[91,2] = PR[90,2] + -20.446;
   1:  PR[91,3] = PR[90,3] + 67.705;
   1:L PR[91] R[100]mm/sec CNT100;
   1:  PR[91,1] = PR[90,1] + -11.459;
   1:  PR[91,2] = PR[90,2] + -21.177;
   1:  PR[91,3] = PR[90,3] + 67.715;
   1:L PR[91] R[100]mm/sec CNT100;
   1:  PR[91,1] = PR[90,1] + -10.164;
   1:  PR[91,2] = PR[90,2] + -21.808;
   1:  PR[91,3] = PR[90,3] + 67.728;
   1:L PR[91] R[100]mm/sec CNT100;
   1:  PR[91,1] = PR[90,1] + -8.831;
   1:  PR[91,2] = PR[90,2] + -22.364;
   1:  PR[91,3] = PR[90,3] + 67.740;
   1:L PR[91] R[100]mm/sec CNT100;
   1:  PR[91,1] = PR[90,1] + -7.465;
   1:  PR[91,2] = PR[90,2] + -22.840;
   1:  PR[91,3] = PR[90,3] + 67.753;
   1:L PR[91] R[100]mm/sec CNT100;
   1:  PR[91,1] = PR[90,1] + -6.953;
   1:  PR[91,2] = PR[90,2] + -22.996;
   1:  PR[91,3] = PR[90,3] + 67.765;
   1:L PR[91] R[100]mm/sec CNT100;
   1:  PR[91,1] = PR[90,1] + -5.836;
   1:  PR[91,2] = PR[90,2] + -23.292;
   1:  PR[91,3] = PR[90,3] + 67.770;
   1:L PR[91] R[100]mm/sec CNT100;
   1:  PR[91,1] = PR[90,1] + -4.672;
   1:  PR[91,2] = PR[90,2] + -23.543;
   1:  PR[91,3] = PR[90,3] + 67.780;
   1:L PR[91] R[100]mm/sec CNT100;
   1:  PR[91,1] = PR[90,1] + -3.852;
   1:  PR[91,2] = PR[90,2] + -23.684;
   1:  PR[91,3] = PR[90,3] + 67.790;
   1:L PR[91] R[100]mm/sec CNT100;
   1:  PR[91,1] = PR[90,1] + -2.746;
   1:  PR[91,2] = PR[90,2] + -23.827;
   1:  PR[91,3] = PR[90,3] + 67.798;
   1:L PR[91] R[100]mm/sec CNT100;
   1:  PR[91,1] = PR[90,1] + -1.556;
   1:  PR[91,2] = PR[90,2] + -23.930;
   1:  PR[91,3] = PR[90,3] + 67.807;
   1:L PR[91] R[100]mm/sec CNT100;
   1:  PR[91,1] = PR[90,1] + -0.980;
   1:  PR[91,2] = PR[90,2] + -23.957;
   1:  PR[91,3] = PR[90,3] + 67.818;
   1:L PR[91] R[100]mm/sec CNT100;
   1:  PR[91,1] = PR[90,1] + -0.123;
   1:  PR[91,2] = PR[90,2] + -23.972;
   1:  PR[91,3] = PR[90,3] + 67.823;
   1:L PR[91] R[100]mm/sec CNT100;
   1:  PR[91] = PR[90];
   1:  PR[91,1] = PR[90,1] + 1.350;
   1:  PR[91,2] = PR[90,2] + -23.928;
   1:  PR[91,3] = PR[90,3] + 69.160;
   1:L PR[91] R[100]mm/sec CNT100;
   1:  PR[91,1] = PR[90,1] + 1.865;
   1:  PR[91,2] = PR[90,2] + -23.891;
   1:  PR[91,3] = PR[90,3] + 67.842;
   1:L PR[91] R[100]mm/sec CNT100;
   1:  PR[91,1] = PR[90,1] + 2.803;
   1:  PR[91,2] = PR[90,2] + -23.796;
   1:  PR[91,3] = PR[90,3] + 67.847;
   1:L PR[91] R[100]mm/sec CNT100;
   1:  PR[91,1] = PR[90,1] + 4.257;
   1:  PR[91,2] = PR[90,2] + -23.576;
   1:  PR[91,3] = PR[90,3] + 67.855;
   1:L PR[91] R[100]mm/sec CNT100;
   1:  PR[91,1] = PR[90,1] + 4.777;
   1:  PR[91,2] = PR[90,2] + -23.476;
   1:  PR[91,3] = PR[90,3] + 67.868;
   1:L PR[91] R[100]mm/sec CNT100;
   1:  PR[91,1] = PR[90,1] + 5.751;
   1:  PR[91,2] = PR[90,2] + -23.255;
   1:  PR[91,3] = PR[90,3] + 67.872;
   1:L PR[91] R[100]mm/sec CNT100;
   1:  PR[91,1] = PR[90,1] + 7.171;
   1:  PR[91,2] = PR[90,2] + -22.858;
   1:  PR[91,3] = PR[90,3] + 67.881;
   1:L PR[91] R[100]mm/sec CNT100;
   1:  PR[91,1] = PR[90,1] + 7.752;
   1:  PR[91,2] = PR[90,2] + -22.667;
   1:  PR[91,3] = PR[90,3] + 67.894;
   1:L PR[91] R[100]mm/sec CNT100;
   1:  PR[91,1] = PR[90,1] + 8.545;
   1:  PR[91,2] = PR[90,2] + -22.382;
   1:  PR[91,3] = PR[90,3] + 67.899;
   1:L PR[91] R[100]mm/sec CNT100;
   1:  PR[91,1] = PR[90,1] + 9.843;
   1:  PR[91,2] = PR[90,2] + -21.845;
   1:  PR[91,3] = PR[90,3] + 67.906;
   1:L PR[91] R[100]mm/sec CNT100;
   1:  PR[91,1] = PR[90,1] + 10.650;
   1:  PR[91,2] = PR[90,2] + -21.467;
   1:  PR[91,3] = PR[90,3] + 67.918;
   1:L PR[91] R[100]mm/sec CNT100;
   1:  PR[91,1] = PR[90,1] + 11.277;
   1:  PR[91,2] = PR[90,2] + -21.146;
   1:  PR[91,3] = PR[90,3] + 67.926;
   1:L PR[91] R[100]mm/sec CNT100;
   1:  PR[91,1] = PR[90,1] + 12.495;
   1:  PR[91,2] = PR[90,2] + -20.458;
   1:  PR[91,3] = PR[90,3] + 67.932;
   1:L PR[91] R[100]mm/sec CNT100;
   1:  PR[91,1] = PR[90,1] + 13.786;
   1:  PR[91,2] = PR[90,2] + -19.621;
   1:  PR[91,3] = PR[90,3] + 67.944;
   1:L PR[91] R[100]mm/sec CNT100;
   1:  PR[91,1] = PR[90,1] + 14.907;
   1:  PR[91,2] = PR[90,2] + -18.796;
   1:  PR[91,3] = PR[90,3] + 67.958;
   1:L PR[91] R[100]mm/sec CNT100;
   1:  PR[91,1] = PR[90,1] + 16.039;
   1:  PR[91,2] = PR[90,2] + -17.854;
   1:  PR[91,3] = PR[90,3] + 67.970;
   1:L PR[91] R[100]mm/sec CNT100;
   1:  PR[91,1] = PR[90,1] + 16.498;
   1:  PR[91,2] = PR[90,2] + -17.439;
   1:  PR[91,3] = PR[90,3] + 67.983;
   1:L PR[91] R[100]mm/sec CNT100;
   1:  PR[91,1] = PR[90,1] + 17.155;
   1:  PR[91,2] = PR[90,2] + -16.805;
   1:  PR[91,3] = PR[90,3] + 67.988;
   1:L PR[91] R[100]mm/sec CNT100;
   1:  PR[91,1] = PR[90,1] + 18.164;
   1:  PR[91,2] = PR[90,2] + -15.730;
   1:  PR[91,3] = PR[90,3] + 67.996;
   1:L PR[91] R[100]mm/sec CNT100;
   1:  PR[91,1] = PR[90,1] + 19.109;
   1:  PR[91,2] = PR[90,2] + -14.593;
   1:  PR[91,3] = PR[90,3] + 68.009;
   1:L PR[91] R[100]mm/sec CNT100;
   1:  PR[91,1] = PR[90,1] + 19.474;
   1:  PR[91,2] = PR[90,2] + -14.114;
   1:  PR[91,3] = PR[90,3] + 68.022;
   1:L PR[91] R[100]mm/sec CNT100;
   1:  PR[91,1] = PR[90,1] + 19.973;
   1:  PR[91,2] = PR[90,2] + -13.416;
   1:  PR[91,3] = PR[90,3] + 68.027;
   1:L PR[91] R[100]mm/sec CNT100;
   1:  PR[91,1] = PR[90,1] + 20.735;
   1:  PR[91,2] = PR[90,2] + -12.238;
   1:  PR[91,3] = PR[90,3] + 68.034;
   1:L PR[91] R[100]mm/sec CNT100;
   1:  PR[91,1] = PR[90,1] + 21.496;
   1:  PR[91,2] = PR[90,2] + -10.892;
   1:  PR[91,3] = PR[90,3] + 68.046;
   1:L PR[91] R[100]mm/sec CNT100;
   1:  PR[91,1] = PR[90,1] + 22.109;
   1:  PR[91,2] = PR[90,2] + -9.634;
   1:  PR[91,3] = PR[90,3] + 68.060;
   1:L PR[91] R[100]mm/sec CNT100;
   1:  PR[91,1] = PR[90,1] + 22.393;
   1:  PR[91,2] = PR[90,2] + -8.982;
   1:  PR[91,3] = PR[90,3] + 68.072;
   1:L PR[91] R[100]mm/sec CNT100;
   1:  PR[91,1] = PR[90,1] + 22.699;
   1:  PR[91,2] = PR[90,2] + -8.213;
   1:  PR[91,3] = PR[90,3] + 68.078;
   1:L PR[91] R[100]mm/sec CNT100;
   1:  PR[91,1] = PR[90,1] + 23.179;
   1:  PR[91,2] = PR[90,2] + -6.820;
   1:  PR[91,3] = PR[90,3] + 68.085;
   1:L PR[91] R[100]mm/sec CNT100;
   1:  PR[91,1] = PR[90,1] + 23.573;
   1:  PR[91,2] = PR[90,2] + -5.402;
   1:  PR[91,3] = PR[90,3] + 68.098;
   1:L PR[91] R[100]mm/sec CNT100;
   1:  PR[91,1] = PR[90,1] + 23.882;
   1:  PR[91,2] = PR[90,2] + -3.962;
   1:  PR[91,3] = PR[90,3] + 68.111;
   1:L PR[91] R[100]mm/sec CNT100;
   1:  PR[91,1] = PR[90,1] + 24.103;
   1:  PR[91,2] = PR[90,2] + -2.511;
   1:  PR[91,3] = PR[90,3] + 68.124;
   1:L PR[91] R[100]mm/sec CNT100;
   1:  PR[91,1] = PR[90,1] + 24.230;
   1:  PR[91,2] = PR[90,2] + -1.123;
   1:  PR[91,3] = PR[90,3] + 68.136;
   1:L PR[91] R[100]mm/sec CNT100;
   1:  PR[91,1] = PR[90,1] + 24.279;
   1:  PR[91,2] = PR[90,2] + 0.502;
   1:  PR[91,3] = PR[90,3] + 68.148;
   1:L PR[91] R[100]mm/sec CNT100;
   1:  PR[91,1] = PR[90,1] + 24.235;
   1:  PR[91,2] = PR[90,2] + 1.903;
   1:  PR[91,3] = PR[90,3] + 68.163;
   1:L PR[91] R[100]mm/sec CNT100;
   1:  PR[91,1] = PR[90,1] + 24.103;
   1:  PR[91,2] = PR[90,2] + 3.366;
   1:  PR[91,3] = PR[90,3] + 68.175;
   1:L PR[91] R[100]mm/sec CNT100;
   1:  PR[91,1] = PR[90,1] + 23.868;
   1:  PR[91,2] = PR[90,2] + 4.890;
   1:  PR[91,3] = PR[90,3] + 68.187;
   1:L PR[91] R[100]mm/sec CNT100;
   1:  PR[91,1] = PR[90,1] + 23.574;
   1:  PR[91,2] = PR[90,2] + 6.257;
   1:  PR[91,3] = PR[90,3] + 68.201;
   1:L PR[91] R[100]mm/sec CNT100;
   1:  PR[91,1] = PR[90,1] + 23.179;
   1:  PR[91,2] = PR[90,2] + 7.675;
   1:  PR[91,3] = PR[90,3] + 68.213;
   1:L PR[91] R[100]mm/sec CNT100;
   1:  PR[91,1] = PR[90,1] + 22.699;
   1:  PR[91,2] = PR[90,2] + 9.068;
   1:  PR[91,3] = PR[90,3] + 68.226;
   1:L PR[91] R[100]mm/sec CNT100;
   1:  PR[91,1] = PR[90,1] + 22.393;
   1:  PR[91,2] = PR[90,2] + 9.837;
   1:  PR[91,3] = PR[90,3] + 68.239;
   1:L PR[91] R[100]mm/sec CNT100;
   1:  PR[91,1] = PR[90,1] + 22.109;
   1:  PR[91,2] = PR[90,2] + 10.489;
   1:  PR[91,3] = PR[90,3] + 68.246;
   1:L PR[91] R[100]mm/sec CNT100;
   1:  PR[91,1] = PR[90,1] + 21.496;
   1:  PR[91,2] = PR[90,2] + 11.748;
   1:  PR[91,3] = PR[90,3] + 68.252;
   1:L PR[91] R[100]mm/sec CNT100;
   1:  PR[91,1] = PR[90,1] + 20.773;
   1:  PR[91,2] = PR[90,2] + 13.030;
   1:  PR[91,3] = PR[90,3] + 68.264;
   1:L PR[91] R[100]mm/sec CNT100;
   1:  PR[91,1] = PR[90,1] + 19.973;
   1:  PR[91,2] = PR[90,2] + 14.271;
   1:  PR[91,3] = PR[90,3] + 68.277;
   1:L PR[91] R[100]mm/sec CNT100;
   1:  PR[91,1] = PR[90,1] + 19.474;
   1:  PR[91,2] = PR[90,2] + 14.969;
   1:  PR[91,3] = PR[90,3] + 68.290;
   1:L PR[91] R[100]mm/sec CNT100;
   1:  PR[91,1] = PR[90,1] + 19.063;
   1:  PR[91,2] = PR[90,2] + 15.506;
   1:  PR[91,3] = PR[90,3] + 68.297;
   1:L PR[91] R[100]mm/sec CNT100;
   1:  PR[91,1] = PR[90,1] + 18.164;
   1:  PR[91,2] = PR[90,2] + 16.585;
   1:  PR[91,3] = PR[90,3] + 68.303;
   1:L PR[91] R[100]mm/sec CNT100;
   1:  PR[91,1] = PR[90,1] + 17.155;
   1:  PR[91,2] = PR[90,2] + 17.660;
   1:  PR[91,3] = PR[90,3] + 68.315;
   1:L PR[91] R[100]mm/sec CNT100;
   1:  PR[91,1] = PR[90,1] + 16.498;
   1:  PR[91,2] = PR[90,2] + 18.294;
   1:  PR[91,3] = PR[90,3] + 68.328;
   1:L PR[91] R[100]mm/sec CNT100;
   1:  PR[91,1] = PR[90,1] + 16.039;
   1:  PR[91,2] = PR[90,2] + 18.710;
   1:  PR[91,3] = PR[90,3] + 68.336;
   1:L PR[91] R[100]mm/sec CNT100;
   1:  PR[91,1] = PR[90,1] + 14.963;
   1:  PR[91,2] = PR[90,2] + 19.607;
   1:  PR[91,3] = PR[90,3] + 68.341;
   1:L PR[91] R[100]mm/sec CNT100;
   1:  PR[91,1] = PR[90,1] + 13.583;
   1:  PR[91,2] = PR[90,2] + 20.617;
   1:  PR[91,3] = PR[90,3] + 68.353;
   1:L PR[91] R[100]mm/sec CNT100;
   1:  PR[91,1] = PR[90,1] + 12.497;
   1:  PR[91,2] = PR[90,2] + 21.312;
   1:  PR[91,3] = PR[90,3] + 68.368;
   1:L PR[91] R[100]mm/sec CNT100;
   1:  PR[91,1] = PR[90,1] + 11.215;
   1:  PR[91,2] = PR[90,2] + 22.035;
   1:  PR[91,3] = PR[90,3] + 68.379;
   1:L PR[91] R[100]mm/sec CNT100;
   1:  PR[91,1] = PR[90,1] + 10.651;
   1:  PR[91,2] = PR[90,2] + 22.322;
   1:  PR[91,3] = PR[90,3] + 68.392;
   1:L PR[91] R[100]mm/sec CNT100;
   1:  PR[91,1] = PR[90,1] + 9.908;
   1:  PR[91,2] = PR[90,2] + 22.672;
   1:  PR[91,3] = PR[90,3] + 68.398;
   1:L PR[91] R[100]mm/sec CNT100;
   1:  PR[91,1] = PR[90,1] + 8.545;
   1:  PR[91,2] = PR[90,2] + 23.237;
   1:  PR[91,3] = PR[90,3] + 68.405;
   1:L PR[91] R[100]mm/sec CNT100;
   1:  PR[91,1] = PR[90,1] + 7.753;
   1:  PR[91,2] = PR[90,2] + 23.523;
   1:  PR[91,3] = PR[90,3] + 68.418;
   1:L PR[91] R[100]mm/sec CNT100;
   1:  PR[91,1] = PR[90,1] + 7.103;
   1:  PR[91,2] = PR[90,2] + 23.734;
   1:  PR[91,3] = PR[90,3] + 68.425;
   1:L PR[91] R[100]mm/sec CNT100;
   1:  PR[91,1] = PR[90,1] + 5.683;
   1:  PR[91,2] = PR[90,2] + 24.127;
   1:  PR[91,3] = PR[90,3] + 68.431;
   1:L PR[91] R[100]mm/sec CNT100;
   1:  PR[91,1] = PR[90,1] + 4.778;
   1:  PR[91,2] = PR[90,2] + 24.331;
   1:  PR[91,3] = PR[90,3] + 68.444;
   1:L PR[91] R[100]mm/sec CNT100;
   1:  PR[91,1] = PR[90,1] + 4.257;
   1:  PR[91,2] = PR[90,2] + 24.432;
   1:  PR[91,3] = PR[90,3] + 68.452;
   1:L PR[91] R[100]mm/sec CNT100;
   1:  PR[91,1] = PR[90,1] + 2.873;
   1:  PR[91,2] = PR[90,2] + 24.643;
   1:  PR[91,3] = PR[90,3] + 68.456;
   1:L PR[91] R[100]mm/sec CNT100;
   1:  PR[91,1] = PR[90,1] + 1.864;
   1:  PR[91,2] = PR[90,2] + 24.746;
   1:  PR[91,3] = PR[90,3] + 68.468;
   1:L PR[91] R[100]mm/sec CNT100;
   1:  PR[91,1] = PR[90,1] + 1.350;
   1:  PR[91,2] = PR[90,2] + 24.783;
   1:  PR[91,3] = PR[90,3] + 68.477;
   1:L PR[91] R[100]mm/sec CNT100;
   1:  PR[91,1] = PR[90,1] + -0.123;
   1:  PR[91,2] = PR[90,2] + 24.827;
   1:  PR[91,3] = PR[90,3] + 68.482;
   1:L PR[91] R[100]mm/sec CNT100;
   1:  PR[91,1] = PR[90,1] + -1.050;
   1:  PR[91,2] = PR[90,2] + 24.809;
   1:  PR[91,3] = PR[90,3] + 68.494;
   1:L PR[91] R[100]mm/sec CNT100;
   1:  PR[91,1] = PR[90,1] + -1.577;
   1:  PR[91,2] = PR[90,2] + 24.784;
   1:  PR[91,3] = PR[90,3] + 68.502;
   1:L PR[91] R[100]mm/sec CNT100;
   1:  PR[91,1] = PR[90,1] + -3.048;
   1:  PR[91,2] = PR[90,2] + 24.651;
   1:  PR[91,3] = PR[90,3] + 68.507;
   1:L PR[91] R[100]mm/sec CNT100;
   1:  PR[91,1] = PR[90,1] + -3.966;
   1:  PR[91,2] = PR[90,2] + 24.522;
   1:  PR[91,3] = PR[90,3] + 68.520;
   1:L PR[91] R[100]mm/sec CNT100;
   1:  PR[91,1] = PR[90,1] + -4.554;
   1:  PR[91,2] = PR[90,2] + 24.421;
   1:  PR[91,3] = PR[90,3] + 68.528;
   1:L PR[91] R[100]mm/sec CNT100;
   1:  PR[91,1] = PR[90,1] + -5.996;
   1:  PR[91,2] = PR[90,2] + 24.109;
   1:  PR[91,3] = PR[90,3] + 68.533;
   1:L PR[91] R[100]mm/sec CNT100;
   1:  PR[91,1] = PR[90,1] + -6.945;
   1:  PR[91,2] = PR[90,2] + 23.853;
   1:  PR[91,3] = PR[90,3] + 68.546;
   1:L PR[91] R[100]mm/sec CNT100;
   1:  PR[91,1] = PR[90,1] + -7.398;
   1:  PR[91,2] = PR[90,2] + 23.716;
   1:  PR[91,3] = PR[90,3] + 68.554;
   1:L PR[91] R[100]mm/sec CNT100;
   1:  PR[91,1] = PR[90,1] + -8.789;
   1:  PR[91,2] = PR[90,2] + 23.235;
   1:  PR[91,3] = PR[90,3] + 68.559;
   1:L PR[91] R[100]mm/sec CNT100;
   1:  PR[91,1] = PR[90,1] + -9.846;
   1:  PR[91,2] = PR[90,2] + 22.805;
   1:  PR[91,3] = PR[90,3] + 68.571;
   1:L PR[91] R[100]mm/sec CNT100;
   1:  PR[91,1] = PR[90,1] + -10.136;
   1:  PR[91,2] = PR[90,2] + 22.676;
   1:  PR[91,3] = PR[90,3] + 68.581;
   1:L PR[91] R[100]mm/sec CNT100;
   1:  PR[91,1] = PR[90,1] + -11.520;
   1:  PR[91,2] = PR[90,2] + 21.999;
   1:  PR[91,3] = PR[90,3] + 68.584;
   1:L PR[91] R[100]mm/sec CNT100;
   1:  PR[91,1] = PR[90,1] + -12.734;
   1:  PR[91,2] = PR[90,2] + 21.313;
   1:  PR[91,3] = PR[90,3] + 68.597;
   1:L PR[91] R[100]mm/sec CNT100;
   1:  PR[91,1] = PR[90,1] + -13.967;
   1:  PR[91,2] = PR[90,2] + 20.517;
   1:  PR[91,3] = PR[90,3] + 68.609;
   1:L PR[91] R[100]mm/sec CNT100;
   1:  PR[91,1] = PR[90,1] + -15.149;
   1:  PR[91,2] = PR[90,2] + 19.649;
   1:  PR[91,3] = PR[90,3] + 68.622;
   1:L PR[91] R[100]mm/sec CNT100;
   1:  PR[91,1] = PR[90,1] + -15.713;
   1:  PR[91,2] = PR[90,2] + 19.194;
   1:  PR[91,3] = PR[90,3] + 68.635;
   1:L PR[91] R[100]mm/sec CNT100;
   1:  PR[91,1] = PR[90,1] + -16.323;
   1:  PR[91,2] = PR[90,2] + 18.669;
   1:  PR[91,3] = PR[90,3] + 68.641;
   1:L PR[91] R[100]mm/sec CNT100;
   1:  PR[91,1] = PR[90,1] + -17.396;
   1:  PR[91,2] = PR[90,2] + 17.657;
   1:  PR[91,3] = PR[90,3] + 68.648;
   1:L PR[91] R[100]mm/sec CNT100;
   1:  PR[91,1] = PR[90,1] + -18.357;
   1:  PR[91,2] = PR[90,2] + 16.635;
   1:  PR[91,3] = PR[90,3] + 68.661;
   1:L PR[91] R[100]mm/sec CNT100;
   1:  PR[91,1] = PR[90,1] + -18.656;
   1:  PR[91,2] = PR[90,2] + 16.293;
   1:  PR[91,3] = PR[90,3] + 68.673;
   1:L PR[91] R[100]mm/sec CNT100;
   1:  PR[91,1] = PR[90,1] + -19.297;
   1:  PR[91,2] = PR[90,2] + 15.512;
   1:  PR[91,3] = PR[90,3] + 68.677;
   1:L PR[91] R[100]mm/sec CNT100;
   1:  PR[91,1] = PR[90,1] + -20.213;
   1:  PR[91,2] = PR[90,2] + 14.268;
   1:  PR[91,3] = PR[90,3] + 68.686;
   1:L PR[91] R[100]mm/sec CNT100;
   1:  PR[91,1] = PR[90,1] + -21.012;
   1:  PR[91,2] = PR[90,2] + 13.031;
   1:  PR[91,3] = PR[90,3] + 68.699;
   1:L PR[91] R[100]mm/sec CNT100;
   1:  PR[91,1] = PR[90,1] + -21.734;
   1:  PR[91,2] = PR[90,2] + 11.748;
   1:  PR[91,3] = PR[90,3] + 68.712;
   1:L PR[91] R[100]mm/sec CNT100;
   1:  PR[91,1] = PR[90,1] + -22.376;
   1:  PR[91,2] = PR[90,2] + 10.426;
   1:  PR[91,3] = PR[90,3] + 68.725;
   1:L PR[91] R[100]mm/sec CNT100;
   1:  PR[91,1] = PR[90,1] + -22.912;
   1:  PR[91,2] = PR[90,2] + 9.133;
   1:  PR[91,3] = PR[90,3] + 68.738;
   1:L PR[91] R[100]mm/sec CNT100;
   1:  PR[91,1] = PR[90,1] + -23.418;
   1:  PR[91,2] = PR[90,2] + 7.675;
   1:  PR[91,3] = PR[90,3] + 68.750;
   1:L PR[91] R[100]mm/sec CNT100;
   1:  PR[91,1] = PR[90,1] + -23.812;
   1:  PR[91,2] = PR[90,2] + 6.257;
   1:  PR[91,3] = PR[90,3] + 68.763;
   1:L PR[91] R[100]mm/sec CNT100;
   1:  PR[91,1] = PR[90,1] + -24.121;
   1:  PR[91,2] = PR[90,2] + 4.817;
   1:  PR[91,3] = PR[90,3] + 68.776;
   1:L PR[91] R[100]mm/sec CNT100;
   1:  PR[91,1] = PR[90,1] + -24.341;
   1:  PR[91,2] = PR[90,2] + 3.366;
   1:  PR[91,3] = PR[90,3] + 68.789;
   1:L PR[91] R[100]mm/sec CNT100;
   1:  PR[91,1] = PR[90,1] + -24.468;
   1:  PR[91,2] = PR[90,2] + 1.978;
   1:  PR[91,3] = PR[90,3] + 68.801;
   1:L PR[91] R[100]mm/sec CNT100;
   1:  PR[91,1] = PR[90,1] + -24.518;
   1:  PR[91,2] = PR[90,2] + 0.353;
   1:  PR[91,3] = PR[90,3] + 68.813;
   1:L PR[91] R[100]mm/sec CNT100;
   1:  PR[91,1] = PR[90,1] + -24.474;
   1:  PR[91,2] = PR[90,2] + -1.048;
   1:  PR[91,3] = PR[90,3] + 68.828;
   1:L PR[91] R[100]mm/sec CNT100;
   1:  PR[91,1] = PR[90,1] + -24.341;
   1:  PR[91,2] = PR[90,2] + -2.511;
   1:  PR[91,3] = PR[90,3] + 68.840;
   1:L PR[91] R[100]mm/sec CNT100;
   1:  PR[91,1] = PR[90,1] + -24.107;
   1:  PR[91,2] = PR[90,2] + -4.035;
   1:  PR[91,3] = PR[90,3] + 68.852;
   1:L PR[91] R[100]mm/sec CNT100;
   1:  PR[91,1] = PR[90,1] + -23.812;
   1:  PR[91,2] = PR[90,2] + -5.402;
   1:  PR[91,3] = PR[90,3] + 68.866;
   1:L PR[91] R[100]mm/sec CNT100;
   1:  PR[91,1] = PR[90,1] + -23.416;
   1:  PR[91,2] = PR[90,2] + -6.826;
   1:  PR[91,3] = PR[90,3] + 68.878;
   1:L PR[91] R[100]mm/sec CNT100;
   1:  PR[91,1] = PR[90,1] + -23.399;
   1:  PR[91,2] = PR[90,2] + -6.880;
   1:  PR[91,3] = PR[90,3] + 68.891;
   1:L PR[91] R[100]mm/sec CNT100;
   1:  PR[91,1] = PR[90,1] + -22.939;
   1:  PR[91,2] = PR[90,2] + -8.209;
   1:L PR[91] R[100]mm/sec CNT100;
   1:  PR[91,1] = PR[90,1] + -22.377;
   1:  PR[91,2] = PR[90,2] + -9.570;
   1:  PR[91,3] = PR[90,3] + 68.904;
   1:L PR[91] R[100]mm/sec CNT100;
   1:  PR[91,1] = PR[90,1] + -21.583;
   1:  PR[91,2] = PR[90,2] + -11.176;
   1:  PR[91,3] = PR[90,3] + 68.916;
   1:L PR[91] R[100]mm/sec CNT100;
   1:  PR[91,1] = PR[90,1] + -20.974;
   1:  PR[91,2] = PR[90,2] + -12.237;
   1:  PR[91,3] = PR[90,3] + 68.932;
   1:L PR[91] R[100]mm/sec CNT100;
   1:  PR[91,1] = PR[90,1] + -20.213;
   1:  PR[91,2] = PR[90,2] + -13.413;
   1:  PR[91,3] = PR[90,3] + 68.942;
   1:L PR[91] R[100]mm/sec CNT100;
   1:  PR[91,1] = PR[90,1] + -19.343;
   1:  PR[91,2] = PR[90,2] + -14.599;
   1:  PR[91,3] = PR[90,3] + 68.955;
   1:L PR[91] R[100]mm/sec CNT100;
   1:  PR[91,1] = PR[90,1] + -18.656;
   1:  PR[91,2] = PR[90,2] + -15.438;
   1:  PR[91,3] = PR[90,3] + 68.967;
   1:L PR[91] R[100]mm/sec CNT100;
   1:  PR[91,1] = PR[90,1] + -18.358;
   1:  PR[91,2] = PR[90,2] + -15.780;
   1:  PR[91,3] = PR[90,3] + 68.977;
   1:L PR[91] R[100]mm/sec CNT100;
   1:  PR[91,1] = PR[90,1] + -17.344;
   1:  PR[91,2] = PR[90,2] + -16.854;
   1:  PR[91,3] = PR[90,3] + 68.981;
   1:L PR[91] R[100]mm/sec CNT100;
   1:  PR[91,1] = PR[90,1] + -16.270;
   1:  PR[91,2] = PR[90,2] + -17.861;
   1:  PR[91,3] = PR[90,3] + 68.994;
   1:L PR[91] R[100]mm/sec CNT100;
   1:  PR[91,1] = PR[90,1] + -15.713;
   1:  PR[91,2] = PR[90,2] + -18.338;
   1:  PR[91,3] = PR[90,3] + 69.006;
   1:L PR[91] R[100]mm/sec CNT100;
   1:  PR[91,1] = PR[90,1] + -15.149;
   1:  PR[91,2] = PR[90,2] + -18.794;
   1:  PR[91,3] = PR[90,3] + 69.013;
   1:L PR[91] R[100]mm/sec CNT100;
   1:  PR[91,1] = PR[90,1] + -13.966;
   1:  PR[91,2] = PR[90,2] + -19.662;
   1:  PR[91,3] = PR[90,3] + 69.019;
   1:L PR[91] R[100]mm/sec CNT100;
   1:  PR[91,1] = PR[90,1] + -12.847;
   1:  PR[91,2] = PR[90,2] + -20.388;
   1:  PR[91,3] = PR[90,3] + 69.032;
   1:L PR[91] R[100]mm/sec CNT100;
   1:  PR[91,1] = PR[90,1] + -11.457;
   1:  PR[91,2] = PR[90,2] + -21.178;
   1:  PR[91,3] = PR[90,3] + 69.043;
   1:L PR[91] R[100]mm/sec CNT100;
   1:  PR[91,1] = PR[90,1] + -10.142;
   1:  PR[91,2] = PR[90,2] + -21.818;
   1:  PR[91,3] = PR[90,3] + 69.057;
   1:L PR[91] R[100]mm/sec CNT100;
   1:  PR[91,1] = PR[90,1] + -8.787;
   1:  PR[91,2] = PR[90,2] + -22.380;
   1:  PR[91,3] = PR[90,3] + 69.070;
   1:L PR[91] R[100]mm/sec CNT100;
   1:  PR[91,1] = PR[90,1] + -7.399;
   1:  PR[91,2] = PR[90,2] + -22.861;
   1:  PR[91,3] = PR[90,3] + 69.083;
   1:L PR[91] R[100]mm/sec CNT100;
   1:  PR[91,1] = PR[90,1] + -6.946;
   1:  PR[91,2] = PR[90,2] + -22.998;
   1:  PR[91,3] = PR[90,3] + 69.095;
   1:L PR[91] R[100]mm/sec CNT100;
   1:  PR[91,1] = PR[90,1] + -5.927;
   1:  PR[91,2] = PR[90,2] + -23.270;
   1:  PR[91,3] = PR[90,3] + 69.099;
   1:L PR[91] R[100]mm/sec CNT100;
   1:  PR[91,1] = PR[90,1] + -4.485;
   1:  PR[91,2] = PR[90,2] + -23.578;
   1:  PR[91,3] = PR[90,3] + 69.109;
   1:L PR[91] R[100]mm/sec CNT100;
   1:  PR[91,1] = PR[90,1] + -3.966;
   1:  PR[91,2] = PR[90,2] + -23.667;
   1:  PR[91,3] = PR[90,3] + 69.121;
   1:L PR[91] R[100]mm/sec CNT100;
   1:  PR[91,1] = PR[90,1] + -3.048;
   1:  PR[91,2] = PR[90,2] + -23.796;
   1:  PR[91,3] = PR[90,3] + 69.126;
   1:L PR[91] R[100]mm/sec CNT100;
   1:  PR[91,1] = PR[90,1] + -1.648;
   1:  PR[91,2] = PR[90,2] + -23.923;
   1:  PR[91,3] = PR[90,3] + 69.134;
   1:L PR[91] R[100]mm/sec CNT100;
   1:  PR[91,1] = PR[90,1] + -1.050;
   1:  PR[91,2] = PR[90,2] + -23.954;
   1:  PR[91,3] = PR[90,3] + 69.146;
   1:L PR[91] R[100]mm/sec CNT100;
   1:  PR[91,1] = PR[90,1] + -0.052;
   1:  PR[91,2] = PR[90,2] + -23.971;
   1:  PR[91,3] = PR[90,3] + 69.151;
   1:L PR[91] R[100]mm/sec CNT100;
   1:  PR[91,1] = PR[90,1] + 1.350;
   1:  PR[91,2] = PR[90,2] + -23.928;
   1:  PR[91,3] = PR[90,3] + 69.160;
   1:L PR[91] R[100]mm/sec CNT100;
   1:  PR[91,1] = PR[90,1] + 1.865;
   1:  PR[91,2] = PR[90,2] + -23.891;
   1:L PR[91] R[100]mm/sec CNT100;
   1:  PR[91,1] = PR[90,1] + 2.803;
   1:  PR[91,2] = PR[90,2] + -23.796;
   1:L PR[91] R[100]mm/sec CNT100;
   1:  PR[91,1] = PR[90,1] + 4.257;
   1:  PR[91,2] = PR[90,2] + -23.576;
   1:L PR[91] R[100]mm/sec CNT100;
   1:  PR[91,1] = PR[90,1] + 4.777;
   1:  PR[91,2] = PR[90,2] + -23.476;
   1:L PR[91] R[100]mm/sec CNT100;
   1:  PR[91,1] = PR[90,1] + 5.751;
   1:  PR[91,2] = PR[90,2] + -23.255;
   1:L PR[91] R[100]mm/sec CNT100;
   1:  PR[91,1] = PR[90,1] + 7.171;
   1:  PR[91,2] = PR[90,2] + -22.858;
   1:L PR[91] R[100]mm/sec CNT100;
   1:  PR[91,1] = PR[90,1] + 7.752;
   1:  PR[91,2] = PR[90,2] + -22.667;
   1:L PR[91] R[100]mm/sec CNT100;
   1:  PR[91,1] = PR[90,1] + 8.545;
   1:  PR[91,2] = PR[90,2] + -22.382;
   1:L PR[91] R[100]mm/sec CNT100;
   1:  PR[91,1] = PR[90,1] + 9.843;
   1:  PR[91,2] = PR[90,2] + -21.845;
   1:L PR[91] R[100]mm/sec CNT100;
   1:  PR[91,1] = PR[90,1] + 10.650;
   1:  PR[91,2] = PR[90,2] + -21.467;
   1:L PR[91] R[100]mm/sec CNT100;
   1:  PR[91,1] = PR[90,1] + 11.277;
   1:  PR[91,2] = PR[90,2] + -21.146;
   1:L PR[91] R[100]mm/sec CNT100;
   1:  PR[91,1] = PR[90,1] + 12.495;
   1:  PR[91,2] = PR[90,2] + -20.458;
   1:L PR[91] R[100]mm/sec CNT100;
   1:  PR[91,1] = PR[90,1] + 13.786;
   1:  PR[91,2] = PR[90,2] + -19.621;
   1:L PR[91] R[100]mm/sec CNT100;
   1:  PR[91,1] = PR[90,1] + 14.907;
   1:  PR[91,2] = PR[90,2] + -18.796;
   1:L PR[91] R[100]mm/sec CNT100;
   1:  PR[91,1] = PR[90,1] + 16.039;
   1:  PR[91,2] = PR[90,2] + -17.854;
   1:L PR[91] R[100]mm/sec CNT100;
   1:  PR[91,1] = PR[90,1] + 16.498;
   1:  PR[91,2] = PR[90,2] + -17.439;
   1:L PR[91] R[100]mm/sec CNT100;
   1:  PR[91,1] = PR[90,1] + 17.155;
   1:  PR[91,2] = PR[90,2] + -16.805;
   1:L PR[91] R[100]mm/sec CNT100;
   1:  PR[91,1] = PR[90,1] + 18.164;
   1:  PR[91,2] = PR[90,2] + -15.730;
   1:L PR[91] R[100]mm/sec CNT100;
   1:  PR[91,1] = PR[90,1] + 19.109;
   1:  PR[91,2] = PR[90,2] + -14.593;
   1:L PR[91] R[100]mm/sec CNT100;
   1:  PR[91,1] = PR[90,1] + 19.474;
   1:  PR[91,2] = PR[90,2] + -14.114;
   1:L PR[91] R[100]mm/sec CNT100;
   1:  PR[91,1] = PR[90,1] + 19.973;
   1:  PR[91,2] = PR[90,2] + -13.416;
   1:L PR[91] R[100]mm/sec CNT100;
   1:  PR[91,1] = PR[90,1] + 20.735;
   1:  PR[91,2] = PR[90,2] + -12.238;
   1:L PR[91] R[100]mm/sec CNT100;
   1:  PR[91,1] = PR[90,1] + 21.496;
   1:  PR[91,2] = PR[90,2] + -10.892;
   1:L PR[91] R[100]mm/sec CNT100;
   1:  PR[91,1] = PR[90,1] + 22.109;
   1:  PR[91,2] = PR[90,2] + -9.634;
   1:L PR[91] R[100]mm/sec CNT100;
   1:  PR[91,1] = PR[90,1] + 22.393;
   1:  PR[91,2] = PR[90,2] + -8.982;
   1:L PR[91] R[100]mm/sec CNT100;
   1:  PR[91,1] = PR[90,1] + 22.699;
   1:  PR[91,2] = PR[90,2] + -8.213;
   1:L PR[91] R[100]mm/sec CNT100;
   1:  PR[91,1] = PR[90,1] + 23.179;
   1:  PR[91,2] = PR[90,2] + -6.820;
   1:L PR[91] R[100]mm/sec CNT100;
   1:  PR[91,1] = PR[90,1] + 23.573;
   1:  PR[91,2] = PR[90,2] + -5.402;
   1:L PR[91] R[100]mm/sec CNT100;
   1:  PR[91,1] = PR[90,1] + 23.882;
   1:  PR[91,2] = PR[90,2] + -3.962;
   1:L PR[91] R[100]mm/sec CNT100;
   1:  PR[91,1] = PR[90,1] + 24.103;
   1:  PR[91,2] = PR[90,2] + -2.511;
   1:L PR[91] R[100]mm/sec CNT100;
   1:  PR[91,1] = PR[90,1] + 24.230;
   1:  PR[91,2] = PR[90,2] + -1.123;
   1:L PR[91] R[100]mm/sec CNT100;
   1:  PR[91,1] = PR[90,1] + 24.279;
   1:  PR[91,2] = PR[90,2] + 0.502;
   1:L PR[91] R[100]mm/sec CNT100;
   1:  PR[91,1] = PR[90,1] + 24.235;
   1:  PR[91,2] = PR[90,2] + 1.903;
   1:L PR[91] R[100]mm/sec CNT100;
   1:  PR[91,1] = PR[90,1] + 24.103;
   1:  PR[91,2] = PR[90,2] + 3.366;
   1:L PR[91] R[100]mm/sec CNT100;
   1:  PR[91,1] = PR[90,1] + 23.868;
   1:  PR[91,2] = PR[90,2] + 4.890;
   1:L PR[91] R[100]mm/sec CNT100;
   1:  PR[91,1] = PR[90,1] + 23.574;
   1:  PR[91,2] = PR[90,2] + 6.257;
   1:L PR[91] R[100]mm/sec CNT100;
   1:  PR[91,1] = PR[90,1] + 23.179;
   1:  PR[91,2] = PR[90,2] + 7.675;
   1:L PR[91] R[100]mm/sec CNT100;
   1:  PR[91,1] = PR[90,1] + 22.699;
   1:  PR[91,2] = PR[90,2] + 9.068;
   1:L PR[91] R[100]mm/sec CNT100;
   1:  PR[91,1] = PR[90,1] + 22.393;
   1:  PR[91,2] = PR[90,2] + 9.837;
   1:L PR[91] R[100]mm/sec CNT100;
   1:  PR[91,1] = PR[90,1] + 22.109;
   1:  PR[91,2] = PR[90,2] + 10.489;
   1:L PR[91] R[100]mm/sec CNT100;
   1:  PR[91,1] = PR[90,1] + 21.496;
   1:  PR[91,2] = PR[90,2] + 11.748;
   1:L PR[91] R[100]mm/sec CNT100;
   1:  PR[91,1] = PR[90,1] + 20.773;
   1:  PR[91,2] = PR[90,2] + 13.030;
   1:L PR[91] R[100]mm/sec CNT100;
   1:  PR[91,1] = PR[90,1] + 19.973;
   1:  PR[91,2] = PR[90,2] + 14.271;
   1:L PR[91] R[100]mm/sec CNT100;
   1:  PR[91,1] = PR[90,1] + 19.474;
   1:  PR[91,2] = PR[90,2] + 14.969;
   1:L PR[91] R[100]mm/sec CNT100;
   1:  PR[91,1] = PR[90,1] + 19.063;
   1:  PR[91,2] = PR[90,2] + 15.506;
   1:L PR[91] R[100]mm/sec CNT100;
   1:  PR[91,1] = PR[90,1] + 18.164;
   1:  PR[91,2] = PR[90,2] + 16.585;
   1:L PR[91] R[100]mm/sec CNT100;
   1:  PR[91,1] = PR[90,1] + 17.155;
   1:  PR[91,2] = PR[90,2] + 17.660;
   1:L PR[91] R[100]mm/sec CNT100;
   1:  PR[91,1] = PR[90,1] + 16.498;
   1:  PR[91,2] = PR[90,2] + 18.294;
   1:L PR[91] R[100]mm/sec CNT100;
   1:  PR[91,1] = PR[90,1] + 16.039;
   1:  PR[91,2] = PR[90,2] + 18.710;
   1:L PR[91] R[100]mm/sec CNT100;
   1:  PR[91,1] = PR[90,1] + 14.963;
   1:  PR[91,2] = PR[90,2] + 19.607;
   1:L PR[91] R[100]mm/sec CNT100;
   1:  PR[91,1] = PR[90,1] + 13.583;
   1:  PR[91,2] = PR[90,2] + 20.617;
   1:L PR[91] R[100]mm/sec CNT100;
   1:  PR[91,1] = PR[90,1] + 12.497;
   1:  PR[91,2] = PR[90,2] + 21.312;
   1:L PR[91] R[100]mm/sec CNT100;
   1:  PR[91,1] = PR[90,1] + 11.215;
   1:  PR[91,2] = PR[90,2] + 22.035;
   1:L PR[91] R[100]mm/sec CNT100;
   1:  PR[91,1] = PR[90,1] + 10.651;
   1:  PR[91,2] = PR[90,2] + 22.322;
   1:L PR[91] R[100]mm/sec CNT100;
   1:  PR[91,1] = PR[90,1] + 9.908;
   1:  PR[91,2] = PR[90,2] + 22.672;
   1:L PR[91] R[100]mm/sec CNT100;
   1:  PR[91,1] = PR[90,1] + 8.545;
   1:  PR[91,2] = PR[90,2] + 23.237;
   1:L PR[91] R[100]mm/sec CNT100;
   1:  PR[91,1] = PR[90,1] + 7.753;
   1:  PR[91,2] = PR[90,2] + 23.523;
   1:L PR[91] R[100]mm/sec CNT100;
   1:  PR[91,1] = PR[90,1] + 7.103;
   1:  PR[91,2] = PR[90,2] + 23.734;
   1:L PR[91] R[100]mm/sec CNT100;
   1:  PR[91,1] = PR[90,1] + 5.683;
   1:  PR[91,2] = PR[90,2] + 24.127;
   1:L PR[91] R[100]mm/sec CNT100;
   1:  PR[91,1] = PR[90,1] + 4.778;
   1:  PR[91,2] = PR[90,2] + 24.331;
   1:L PR[91] R[100]mm/sec CNT100;
   1:  PR[91,1] = PR[90,1] + 4.257;
   1:  PR[91,2] = PR[90,2] + 24.432;
   1:L PR[91] R[100]mm/sec CNT100;
   1:  PR[91,1] = PR[90,1] + 2.873;
   1:  PR[91,2] = PR[90,2] + 24.643;
   1:L PR[91] R[100]mm/sec CNT100;
   1:  PR[91,1] = PR[90,1] + 1.864;
   1:  PR[91,2] = PR[90,2] + 24.746;
   1:L PR[91] R[100]mm/sec CNT100;
   1:  PR[91,1] = PR[90,1] + 1.350;
   1:  PR[91,2] = PR[90,2] + 24.783;
   1:L PR[91] R[100]mm/sec CNT100;
   1:  PR[91,1] = PR[90,1] + -0.123;
   1:  PR[91,2] = PR[90,2] + 24.827;
   1:L PR[91] R[100]mm/sec CNT100;
   1:  PR[91,1] = PR[90,1] + -1.050;
   1:  PR[91,2] = PR[90,2] + 24.809;
   1:L PR[91] R[100]mm/sec CNT100;
   1:  PR[91,1] = PR[90,1] + -1.577;
   1:  PR[91,2] = PR[90,2] + 24.784;
   1:L PR[91] R[100]mm/sec CNT100;
   1:  PR[91,1] = PR[90,1] + -3.048;
   1:  PR[91,2] = PR[90,2] + 24.651;
   1:L PR[91] R[100]mm/sec CNT100;
   1:  PR[91,1] = PR[90,1] + -3.966;
   1:  PR[91,2] = PR[90,2] + 24.522;
   1:L PR[91] R[100]mm/sec CNT100;
   1:  PR[91,1] = PR[90,1] + -4.554;
   1:  PR[91,2] = PR[90,2] + 24.421;
   1:L PR[91] R[100]mm/sec CNT100;
   1:  PR[91,1] = PR[90,1] + -5.996;
   1:  PR[91,2] = PR[90,2] + 24.109;
   1:L PR[91] R[100]mm/sec CNT100;
   1:  PR[91,1] = PR[90,1] + -6.945;
   1:  PR[91,2] = PR[90,2] + 23.853;
   1:L PR[91] R[100]mm/sec CNT100;
   1:  PR[91,1] = PR[90,1] + -7.398;
   1:  PR[91,2] = PR[90,2] + 23.716;
   1:L PR[91] R[100]mm/sec CNT100;
   1:  PR[91,1] = PR[90,1] + -8.789;
   1:  PR[91,2] = PR[90,2] + 23.235;
   1:L PR[91] R[100]mm/sec CNT100;
   1:  PR[91,1] = PR[90,1] + -9.846;
   1:  PR[91,2] = PR[90,2] + 22.805;
   1:L PR[91] R[100]mm/sec CNT100;
   1:  PR[91,1] = PR[90,1] + -10.136;
   1:  PR[91,2] = PR[90,2] + 22.676;
   1:L PR[91] R[100]mm/sec CNT100;
   1:  PR[91,1] = PR[90,1] + -11.520;
   1:  PR[91,2] = PR[90,2] + 21.999;
   1:L PR[91] R[100]mm/sec CNT100;
   1:  PR[91,1] = PR[90,1] + -12.734;
   1:  PR[91,2] = PR[90,2] + 21.313;
   1:L PR[91] R[100]mm/sec CNT100;
   1:  PR[91,1] = PR[90,1] + -13.967;
   1:  PR[91,2] = PR[90,2] + 20.517;
   1:L PR[91] R[100]mm/sec CNT100;
   1:  PR[91,1] = PR[90,1] + -15.149;
   1:  PR[91,2] = PR[90,2] + 19.649;
   1:L PR[91] R[100]mm/sec CNT100;
   1:  PR[91,1] = PR[90,1] + -15.713;
   1:  PR[91,2] = PR[90,2] + 19.194;
   1:L PR[91] R[100]mm/sec CNT100;
   1:  PR[91,1] = PR[90,1] + -16.323;
   1:  PR[91,2] = PR[90,2] + 18.669;
   1:L PR[91] R[100]mm/sec CNT100;
   1:  PR[91,1] = PR[90,1] + -17.396;
   1:  PR[91,2] = PR[90,2] + 17.657;
   1:L PR[91] R[100]mm/sec CNT100;
   1:  PR[91,1] = PR[90,1] + -18.357;
   1:  PR[91,2] = PR[90,2] + 16.635;
   1:L PR[91] R[100]mm/sec CNT100;
   1:  PR[91,1] = PR[90,1] + -18.656;
   1:  PR[91,2] = PR[90,2] + 16.293;
   1:L PR[91] R[100]mm/sec CNT100;
   1:  PR[91,1] = PR[90,1] + -19.297;
   1:  PR[91,2] = PR[90,2] + 15.512;
   1:L PR[91] R[100]mm/sec CNT100;
   1:  PR[91,1] = PR[90,1] + -20.213;
   1:  PR[91,2] = PR[90,2] + 14.268;
   1:L PR[91] R[100]mm/sec CNT100;
   1:  PR[91,1] = PR[90,1] + -21.012;
   1:  PR[91,2] = PR[90,2] + 13.031;
   1:L PR[91] R[100]mm/sec CNT100;
   1:  PR[91,1] = PR[90,1] + -21.734;
   1:  PR[91,2] = PR[90,2] + 11.748;
   1:L PR[91] R[100]mm/sec CNT100;
   1:  PR[91,1] = PR[90,1] + -22.376;
   1:  PR[91,2] = PR[90,2] + 10.426;
   1:L PR[91] R[100]mm/sec CNT100;
   1:  PR[91,1] = PR[90,1] + -22.912;
   1:  PR[91,2] = PR[90,2] + 9.133;
   1:L PR[91] R[100]mm/sec CNT100;
   1:  PR[91,1] = PR[90,1] + -23.418;
   1:  PR[91,2] = PR[90,2] + 7.675;
   1:L PR[91] R[100]mm/sec CNT100;
   1:  PR[91,1] = PR[90,1] + -23.812;
   1:  PR[91,2] = PR[90,2] + 6.257;
   1:L PR[91] R[100]mm/sec CNT100;
   1:  PR[91,1] = PR[90,1] + -24.121;
   1:  PR[91,2] = PR[90,2] + 4.817;
   1:L PR[91] R[100]mm/sec CNT100;
   1:  PR[91,1] = PR[90,1] + -24.341;
   1:  PR[91,2] = PR[90,2] + 3.366;
   1:L PR[91] R[100]mm/sec CNT100;
   1:  PR[91,1] = PR[90,1] + -24.468;
   1:  PR[91,2] = PR[90,2] + 1.978;
   1:L PR[91] R[100]mm/sec CNT100;
   1:  PR[91,1] = PR[90,1] + -24.518;
   1:  PR[91,2] = PR[90,2] + 0.353;
   1:L PR[91] R[100]mm/sec CNT100;
   1:  PR[91,1] = PR[90,1] + -24.474;
   1:  PR[91,2] = PR[90,2] + -1.048;
   1:L PR[91] R[100]mm/sec CNT100;
   1:  PR[91,1] = PR[90,1] + -24.341;
   1:  PR[91,2] = PR[90,2] + -2.511;
   1:L PR[91] R[100]mm/sec CNT100;
   1:  PR[91,1] = PR[90,1] + -24.107;
   1:  PR[91,2] = PR[90,2] + -4.035;
   1:L PR[91] R[100]mm/sec CNT100;
   1:  PR[91,1] = PR[90,1] + -23.812;
   1:  PR[91,2] = PR[90,2] + -5.402;
   1:L PR[91] R[100]mm/sec CNT100;
   1:  PR[91,1] = PR[90,1] + -23.416;
   1:  PR[91,2] = PR[90,2] + -6.826;
   1:L PR[91] R[100]mm/sec CNT100;
   1:  PR[91,1] = PR[90,1] + -23.399;
   1:  PR[91,2] = PR[90,2] + -6.880;
   1:L PR[91] R[100]mm/sec CNT100;
   1:  PR[91,1] = PR[90,1] + -22.939;
   1:  PR[91,2] = PR[90,2] + -8.209;
   1:L PR[91] R[100]mm/sec CNT100;
   1:  PR[91,1] = PR[90,1] + -22.377;
   1:  PR[91,2] = PR[90,2] + -9.570;
   1:L PR[91] R[100]mm/sec CNT100;
   1:  PR[91,1] = PR[90,1] + -21.583;
   1:  PR[91,2] = PR[90,2] + -11.176;
   1:L PR[91] R[100]mm/sec CNT100;
   1:  PR[91,1] = PR[90,1] + -20.974;
   1:  PR[91,2] = PR[90,2] + -12.237;
   1:L PR[91] R[100]mm/sec CNT100;
   1:  PR[91,1] = PR[90,1] + -20.213;
   1:  PR[91,2] = PR[90,2] + -13.413;
   1:L PR[91] R[100]mm/sec CNT100;
   1:  PR[91,1] = PR[90,1] + -19.343;
   1:  PR[91,2] = PR[90,2] + -14.599;
   1:L PR[91] R[100]mm/sec CNT100;
   1:  PR[91,1] = PR[90,1] + -18.656;
   1:  PR[91,2] = PR[90,2] + -15.438;
   1:L PR[91] R[100]mm/sec CNT100;
   1:  PR[91,1] = PR[90,1] + -18.358;
   1:  PR[91,2] = PR[90,2] + -15.780;
   1:L PR[91] R[100]mm/sec CNT100;
   1:  PR[91,1] = PR[90,1] + -17.344;
   1:  PR[91,2] = PR[90,2] + -16.854;
   1:L PR[91] R[100]mm/sec CNT100;
   1:  PR[91,1] = PR[90,1] + -16.270;
   1:  PR[91,2] = PR[90,2] + -17.861;
   1:L PR[91] R[100]mm/sec CNT100;
   1:  PR[91,1] = PR[90,1] + -15.713;
   1:  PR[91,2] = PR[90,2] + -18.338;
   1:L PR[91] R[100]mm/sec CNT100;
   1:  PR[91,1] = PR[90,1] + -15.149;
   1:  PR[91,2] = PR[90,2] + -18.794;
   1:L PR[91] R[100]mm/sec CNT100;
   1:  PR[91,1] = PR[90,1] + -13.966;
   1:  PR[91,2] = PR[90,2] + -19.662;
   1:L PR[91] R[100]mm/sec CNT100;
   1:  PR[91,1] = PR[90,1] + -12.847;
   1:  PR[91,2] = PR[90,2] + -20.388;
   1:L PR[91] R[100]mm/sec CNT100;
   1:  PR[91,1] = PR[90,1] + -11.457;
   1:  PR[91,2] = PR[90,2] + -21.178;
   1:L PR[91] R[100]mm/sec CNT100;
   1:  PR[91,1] = PR[90,1] + -10.142;
   1:  PR[91,2] = PR[90,2] + -21.818;
   1:L PR[91] R[100]mm/sec CNT100;
   1:  PR[91,1] = PR[90,1] + -8.787;
   1:  PR[91,2] = PR[90,2] + -22.380;
   1:L PR[91] R[100]mm/sec CNT100;
   1:  PR[91,1] = PR[90,1] + -7.399;
   1:  PR[91,2] = PR[90,2] + -22.861;
   1:L PR[91] R[100]mm/sec CNT100;
   1:  PR[91,1] = PR[90,1] + -6.946;
   1:  PR[91,2] = PR[90,2] + -22.998;
   1:L PR[91] R[100]mm/sec CNT100;
   1:  PR[91,1] = PR[90,1] + -5.927;
   1:  PR[91,2] = PR[90,2] + -23.270;
   1:L PR[91] R[100]mm/sec CNT100;
   1:  PR[91,1] = PR[90,1] + -4.485;
   1:  PR[91,2] = PR[90,2] + -23.578;
   1:L PR[91] R[100]mm/sec CNT100;
   1:  PR[91,1] = PR[90,1] + -3.966;
   1:  PR[91,2] = PR[90,2] + -23.667;
   1:L PR[91] R[100]mm/sec CNT100;
   1:  PR[91,1] = PR[90,1] + -3.048;
   1:  PR[91,2] = PR[90,2] + -23.796;
   1:L PR[91] R[100]mm/sec CNT100;
   1:  PR[91,1] = PR[90,1] + -1.648;
   1:  PR[91,2] = PR[90,2] + -23.923;
   1:L PR[91] R[100]mm/sec CNT100;
   1:  PR[91,1] = PR[90,1] + -1.050;
   1:  PR[91,2] = PR[90,2] + -23.954;
   1:L PR[91] R[100]mm/sec CNT100;
   1:  PR[91,1] = PR[90,1] + -0.052;
   1:  PR[91,2] = PR[90,2] + -23.971;
   1:L PR[91] R[100]mm/sec CNT100 TB   .50sec,CALL END_PUD;
   1:  DO[117:Laser Start]=OFF;
   1:  PR[92] = PR[91];
   1:  PR[92,3] = PR[92,3] + 50;
   1:J PR[92] 10% FINE;
   1:  WAIT   5.00(sec);
   1:  DO[119:Gas]=OFF;
   1:  CALL HOME_ALL;
/POS
/END
